// TIA Portal V16 program export: 6 tag tables, 0 data types, 9 data blocks, 25 code blocks (in call order from the OBs), 17 instance data blocks

VAR_GLOBAL   // PLC tag table "Analógicas"
   FQ301_MEDIDOR_CAUDAL AT %IW16 : Word;
   PC401_SENSOR_PRESSÃO AT %IW18 : Word;
END_VAR

VAR_GLOBAL   // PLC tag table "Default tag table"
   FirstScan AT %M1.0 : Bool;
   FALLING_EDGE_MAN_AUTO AT %M100.0 : Bool;
   RISING_EDGE_ETAPA_6 AT %M100.2 : Bool;
   FALLING_EDGE_BOT_EMERG AT %M100.5 : Bool;
   FALLIN_EDGE_BOT_EMERG_2 AT %M100.6 : Bool;
   FALLING_EDGE_ETAPA_6 AT %M100.7 : Bool;
   MBIT_DISP_1 AT %M101.0 : Bool;
   MBIT_DISP_2 AT %M101.1 : Bool;
   MBIT_DISP_3 AT %M101.2 : Bool;
   MBIT_DISP_4 AT %M101.3 : Bool;
   MBIT_DISP_5 AT %M101.4 : Bool;
   MBIT_DISP_6 AT %M101.5 : Bool;
   MBIT_DISP_7 AT %M101.6 : Bool;
   MBIT_DISP_8 AT %M101.7 : Bool;
   MBIT_DISP_9 AT %M102.0 : Bool;
   MBIT_DISP_10 AT %M102.1 : Bool;
   MBIT_DISP_11 AT %M102.2 : Bool;
   MBIT_DISP_12 AT %M102.3 : Bool;
   MBIT_DISP_13 AT %M102.4 : Bool;
   MBIT_DISP_14 AT %M102.5 : Bool;
   MBIT_DISP_15 AT %M102.6 : Bool;
   MBIT_DISP_16 AT %M102.7 : Bool;
   MBIT_DISP_DIF_3Q1_32 AT %M103.0 : Bool;
   MBIT_DISP_DIF_3Q3 AT %M103.1 : Bool;
   MBIT_DISP_DIF_4Q1_4Q2 AT %M103.2 : Bool;
   MBIT_FALHA_24VDC AT %M103.3 : Bool;
   MBIT_FALHA_220VAC AT %M103.4 : Bool;
   MBIT_FALHA_24VAC AT %M103.5 : Bool;
   RISING_EDGE_ETAPA_55 AT %M103.7 : Bool;
   RISING_EDGE_START_CICLO AT %M104.0 : Bool;
   Tag_1 AT %M200.0 : Bool;
END_VAR

VAR_GLOBAL   // PLC tag table "Estados_Componentes"
   BS001A_ON AT %I1.5 : Bool;
   BS001A_DISPARO AT %I2.0 : Bool;
   BS001B_ON AT %I2.1 : Bool;
   BS001B_DISPARO AT %I2.2 : Bool;
   XV102_ABERTA AT %I2.3 : Bool;
   XV102_FECHADA AT %I2.4 : Bool;
   XV101_ABERTA AT %I2.5 : Bool;
   MX201_ON AT %I2.6 : Bool;
   MX201_DISPARO AT %I2.7 : Bool;
   BH201_ON AT %I3.0 : Bool;
   BH201_DISPARO AT %I3.1 : Bool;
   MX301_ON AT %I3.2 : Bool;
   MX301_DISPARO AT %I3.3 : Bool;
   BM401_ON AT %I3.4 : Bool;
   BM401_DISPARO AT %I3.5 : Bool;
   BS501_ON AT %I3.6 : Bool;
   BS501_DISPARO AT %I3.7 : Bool;
   MX601_ON AT %I4.0 : Bool;
   MX601_DISPARO AT %I4.1 : Bool;
   BD601_ON AT %I4.2 : Bool;
   BD601_DISPARO AT %I4.3 : Bool;
   BD602_ON AT %I4.4 : Bool;
   BD602_DISPARO AT %I4.5 : Bool;
   MX603_ON AT %I4.6 : Bool;
   MX603_DISPARO AT %I4.7 : Bool;
   BD603_ON AT %I5.0 : Bool;
   BD603_DISPARO AT %I5.1 : Bool;
   MX604_ON AT %I5.2 : Bool;
   MX604_DISPARO AT %I5.3 : Bool;
   BD604_ON AT %I5.4 : Bool;
   BD604_DISPARO AT %I5.5 : Bool;
   MX605_ON AT %I5.6 : Bool;
   MX605_DISPARO AT %I5.7 : Bool;
   BD605_ON AT %I6.0 : Bool;
   BD605_DISPARO AT %I6.1 : Bool;
   BOT_EMERGÊNCIA AT %I6.2 : Bool;
   PH201_CONT_PH AT %I6.3 : Bool;
   PH301_CONT_PH AT %I6.4 : Bool;
   TEMPERATURA_ATINGIDA AT %I6.5 : Bool;
   RH201_CONT_REDOX AT %I6.6 : Bool;
END_VAR

VAR_GLOBAL   // PLC tag table "Falhas"
   DISPARO_DIF_3Q1_32 AT %I0.0 : Bool;
   DISPARO_DIFERENCIAL_3Q3 AT %I0.1 : Bool;
   DISPARO_DIFERENCIAL_4Q1_4Q2 AT %I0.2 : Bool;
   FALHA_24VDC AT %I0.3 : Bool;
   FALHA_220VAC AT %I0.4 : Bool;
   FALHA_24VAC AT %I0.5 : Bool;
END_VAR

VAR_GLOBAL   // PLC tag table "Níveis"
   LSH001_TK00 AT %I0.6 : Bool;
   LSL001_TK00 AT %I1.0 : Bool;
   LSH501_TK05 AT %I1.3 : Bool;
   LSL501_TK05 AT %I1.4 : Bool;
   LSH101_TK01 AT %I1.1 : Bool;
   LS201_TK02 AT %IW12 : Word;
   LS301_TK03 AT %IW14 : Word;
   LSL101_TK01 AT %I1.2 : Bool;
   LSM001_TK00 AT %I0.7 : Bool;
END_VAR

VAR_GLOBAL   // PLC tag table "Saídas"
   BS001A AT %Q0.0 : Bool;
   BS001B AT %Q0.1 : Bool;
   XV101 AT %Q3.3 : Bool;
   XV102 AT %Q3.4 : Bool;
   MX201 AT %Q0.4 : Bool;
   BH201 AT %Q0.5 : Bool;
   MX301 AT %Q0.6 : Bool;
   ALIM_BM401 AT %Q0.7 : Bool;
   LIGAR_BM401 AT %Q3.1 : Bool;
   BS501 AT %Q1.1 : Bool;
   MX601 AT %Q2.0 : Bool;
   BD601 AT %Q2.1 : Bool;
   BD602 AT %Q2.2 : Bool;
   MX603 AT %Q2.3 : Bool;
   BD603 AT %Q2.4 : Bool;
   MX604 AT %Q2.5 : Bool;
   BD604 AT %Q2.6 : Bool;
   MX605 AT %Q2.7 : Bool;
   BD605 AT %Q0.2 : Bool;
   ALARME AT %Q3.2 : Bool;
END_VAR

DATA_BLOCK "Alarmes"   // DB13
{ S7_Optimized_Access := 'TRUE' }
VERSION : 0.1
// stored: AutoNumber true, IsOnlyStoredInLoadMemory false, IsRetainMemResEnabled false, IsWriteProtectedInAS false, MemoryReserve 100
   VAR
      ALARMES_1 : Word;
      ALARMES_2 : Word;
      ALARME_DISPARO : Bool;
      PRESSÃO_MÁX : Bool;
      XV102_NÃO_ABRIU : Bool;
      XV102_NÃO_FECHOU : Bool;
   END_VAR
   VAR RETAIN
      TEMP_ABERT_XV102 : Time;
      TEMP_FECHO_XV102 : Time;
   END_VAR
BEGIN
END_DATA_BLOCK

DATA_BLOCK "Info_Ciclo"   // DB10
{ S7_Optimized_Access := 'TRUE' }
VERSION : 0.1
// stored: AutoNumber true, IsOnlyStoredInLoadMemory false, IsRetainMemResEnabled false, IsWriteProtectedInAS false, MemoryReserve 100
   VAR RETAIN
      LS101_SR : Bool;
   END_VAR
   VAR
      ESTADO_CICLO : Bool;
      CONTAGEM_CICLOS : Int;
      LIMITE_CONTAGEM : Bool;
   END_VAR
BEGIN
END_DATA_BLOCK

DATA_BLOCK "Analógicas"   // DB12
{ S7_Optimized_Access := 'TRUE' }
VERSION : 0.1
// stored: AutoNumber true, IsOnlyStoredInLoadMemory false, IsRetainMemResEnabled false, IsWriteProtectedInAS false, MemoryReserve 100
   VAR
      CAUDAL_FQ301 : Real;
      PRESSÃO_PC401 : Real;
   END_VAR
BEGIN
END_DATA_BLOCK

DATA_BLOCK "Estados_HMI_DB"   // DB15
{ S7_Optimized_Access := 'TRUE' }
VERSION : 0.1
// stored: AutoNumber true, IsOnlyStoredInLoadMemory false, IsRetainMemResEnabled false, IsWriteProtectedInAS false, MemoryReserve 100
   VAR
      MX201 : Bool;
      MX601 : Bool;
      XV101 : Bool;
      XV102 : Bool;
      BD601 : Bool;
      BD602 : Bool;
      BH201 : Bool;
      PH201 : Bool;
      RH201 : Bool;
      MX603 : Bool;
      BD603 : Bool;
      MX301 : Bool;
      PH301 : Bool;
      BM401 : Bool;
      MX604 : Bool;
      BD604 : Bool;
      MX605 : Bool;
      BD605 : Bool;
      BS001A : Bool;
      BS001B : Bool;
      BS501 : Bool;
      T_ATUAL_AREJAMENTO : Time;
      T_ATUAL_REDUÇÃO : Time;
      T_ATUAL_PRECIPITAÇÃO : Time;
      T_ATUAL_ALARME_PC401 : Time;
      T_ATUAL_COAG : Time;
      T_ATUAL_HISTERESE : Time;
   END_VAR
BEGIN
END_DATA_BLOCK

DATA_BLOCK "Inputs_HMI"   // DB14
{ S7_Optimized_Access := 'TRUE' }
VERSION : 0.1
// stored: AutoNumber true, IsOnlyStoredInLoadMemory false, IsRetainMemResEnabled false, IsWriteProtectedInAS false, MemoryReserve 100
   VAR RETAIN
      MODO_1 : Bool;
      MODO_2 : Bool;
   END_VAR
   VAR
      RESET_ALARME : Bool;
      START_CICLO : Bool;
   END_VAR
   VAR RETAIN
      MAN_AUTO : Bool;
   END_VAR
   VAR
      ON_OFF_MX201 : Bool;
      ON_OFF_MX301 : Bool;
      ON_OFF_MX601 : Bool;
      ON_OFF_MX603 : Bool;
      ON_OFF_MX604 : Bool;
      ON_OFF_MX605 : Bool;
      ON_OFF_BD601 : Bool;
      ON_OFF_BD602 : Bool;
      ON_OFF_BD603 : Bool;
      ON_OFF_BD604 : Bool;
      ON_OFF_BD605 : Bool;
      ON_OFF_BS001A : Bool;
      ON_OFF_BS001B : Bool;
      ON_OFF_BS501 : Bool;
      ON_OFF_BH201 : Bool;
      ON_OFF_BM401 : Bool;
      ON_OFF_XV101 : Bool;
      ON_OFF_XV102 : Bool;
   END_VAR
   VAR RETAIN
      TEMP_AREJAMENTO : Time := T#0m;
      TEMP_REDUÇÃO : Time := T#0m;
      TEMP_PRECIPITAÇÃO : Time := T#0m;
      TEMP_ALARME : Time := T#0m;
      TEMP_DOS_COAG : Time;
      HISTERESE : Time;
      SETPOINT_PC401 : Real;
      SP_LSH_TK02 : Real;
      SP_LSM_TK02 : Real;
      SP_LSL_TK02 : Real;
      SP_LSH_TK03 : Real;
      SP_LSM_TK03 : Real;
      SP_LSL_TK03 : Real;
   END_VAR
   VAR
      SALTAR_HISTERESE : Bool;
      RESET_CONT_CICLOS : Bool;
   END_VAR
   VAR RETAIN
      ENABLE_DISABLE_BD603 : Bool := true;
      SUSPENSÃO_CICLO_PRENSA : Bool;
      IGNORAR_LSH101_LSH501 : Bool;
   END_VAR
BEGIN
END_DATA_BLOCK

DATA_BLOCK "Níveis_TK02_TK03"   // DB11
{ S7_Optimized_Access := 'TRUE' }
VERSION : 0.1
// stored: AutoNumber true, IsOnlyStoredInLoadMemory false, IsRetainMemResEnabled false, IsWriteProtectedInAS false, MemoryReserve 100
   VAR
      LSH301 : Bool;
      LSM301 : Bool;
   END_VAR
   VAR RETAIN
      LSL301 : Bool;
   END_VAR
   VAR
      LSH201 : Bool;
      LSM201 : Bool;
      LSL201 : Bool;
      NÍVEL_EM_METROS_TK03 : Real;
      NÍVEL_EM_METROS_TK02 : Real;
   END_VAR
BEGIN
END_DATA_BLOCK

DATA_BLOCK "Etapas_Grafcet_1"   // DB4
{ S7_Optimized_Access := 'TRUE' }
VERSION : 0.1
// stored: AutoNumber true, IsOnlyStoredInLoadMemory false, IsRetainMemResEnabled false, IsWriteProtectedInAS false, MemoryReserve 100
   VAR RETAIN
      ETAPA_1 : Bool;
      ETAPA_2 : Bool;
      ETAPA_3 : Bool;
      ETAPA_4 : Bool;
      ETAPA_5 : Bool;
      ETAPA_6 : Bool;
      ETAPA_7 : Bool;
      ETAPA_8 : Bool;
      ETAPA_9 : Bool;
      ETAPA_33 : Bool;
      ETAPA_55 : Bool;
      RESET_ETAPA_1 : Bool;
      SUSPENSÃO_CICLO : Bool;
   END_VAR
BEGIN
END_DATA_BLOCK

DATA_BLOCK "Etapas_Grafcet_2"   // DB1
{ S7_Optimized_Access := 'TRUE' }
VERSION : 0.1
// stored: AutoNumber true, IsOnlyStoredInLoadMemory false, IsRetainMemResEnabled false, IsWriteProtectedInAS false, MemoryReserve 100
   VAR RETAIN
      ETAPA_10 : Bool;
      ETAPA_11 : Bool;
      ETAPA_12 : Bool;
      RESET_ETAPA_10 : Bool;
   END_VAR
BEGIN
END_DATA_BLOCK

DATA_BLOCK "Etapas_Grafcet_3"   // DB3
{ S7_Optimized_Access := 'TRUE' }
VERSION : 0.1
// stored: AutoNumber true, IsOnlyStoredInLoadMemory false, IsRetainMemResEnabled false, IsWriteProtectedInAS false, MemoryReserve 100
   VAR RETAIN
      ETAPA_13 : Bool;
      ETAPA_14 : Bool;
      ETAPA_15 : Bool;
      RESET_ETAPA_13 : Bool;
   END_VAR
BEGIN
END_DATA_BLOCK

ORGANIZATION_BLOCK "Main"   // OB1, LAD, ProgramCycle
TITLE = "Main Program Sweep (Cycle)"
{ S7_Optimized_Access := 'TRUE' }
VERSION : 0.1
// stored: AutoNumber true, IsIECCheckEnabled false, SetENOAutomatically false
BEGIN

REGION Network 1: Alimentação ao processo
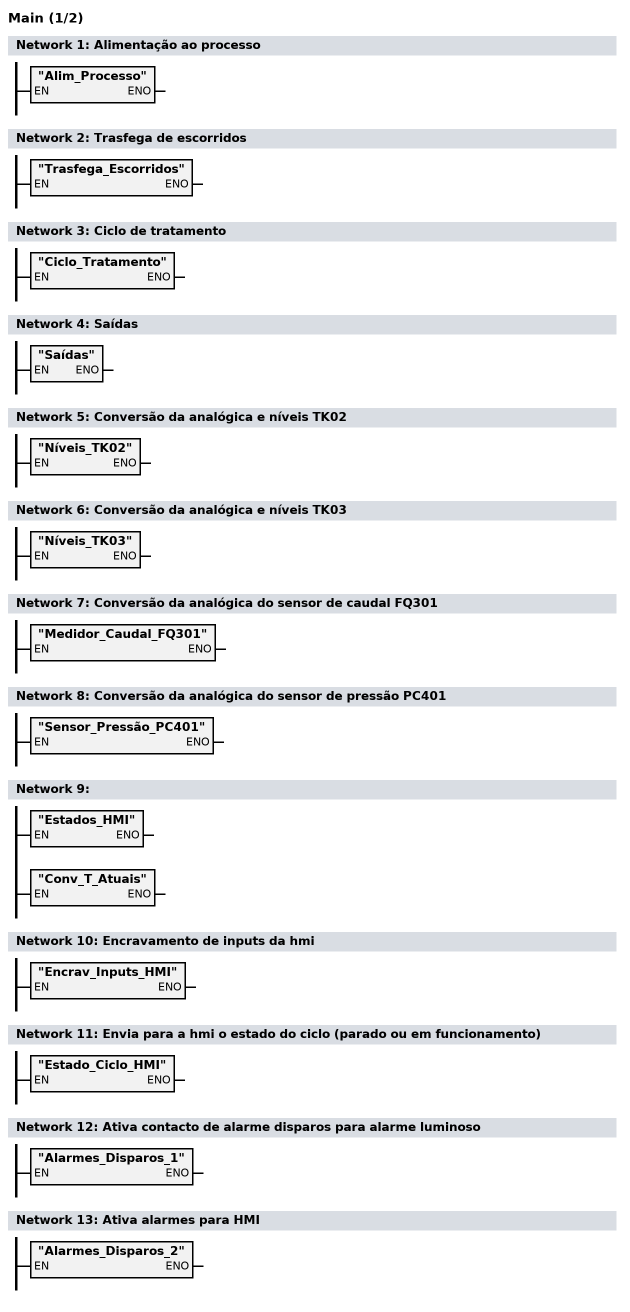
   RUNG wire#powerrail
      "Alim_Processo"()
   END_RUNG
   // the same network as SCL:
   "Alim_Processo"();
END_REGION

REGION Network 2: Trasfega de escorridos
   RUNG wire#powerrail
      "Trasfega_Escorridos"()
   END_RUNG
   // the same network as SCL:
   "Trasfega_Escorridos"();
END_REGION

REGION Network 3: Ciclo de tratamento
   RUNG wire#powerrail
      "Ciclo_Tratamento"()
   END_RUNG
   // the same network as SCL:
   "Ciclo_Tratamento"();
END_REGION

REGION Network 4: Saídas
   RUNG wire#powerrail
      "Saídas"()
   END_RUNG
   // the same network as SCL:
   "Saídas"();
END_REGION

REGION Network 5: Conversão da analógica e níveis TK02
   RUNG wire#powerrail
      "Níveis_TK02"()
   END_RUNG
   // the same network as SCL:
   "Níveis_TK02"();
END_REGION

REGION Network 6: Conversão da analógica e níveis TK03
   RUNG wire#powerrail
      "Níveis_TK03"()
   END_RUNG
   // the same network as SCL:
   "Níveis_TK03"();
END_REGION

REGION Network 7: Conversão da analógica do sensor de caudal FQ301
   RUNG wire#powerrail
      "Medidor_Caudal_FQ301"()
   END_RUNG
   // the same network as SCL:
   "Medidor_Caudal_FQ301"();
END_REGION

REGION Network 8: Conversão da analógica do sensor de pressão PC401
   RUNG wire#powerrail
      "Sensor_Pressão_PC401"()
   END_RUNG
   // the same network as SCL:
   "Sensor_Pressão_PC401"();
END_REGION

REGION Network 9
   RUNG wire#powerrail
      "Estados_HMI"()
   END_RUNG
   RUNG wire#powerrail
      "Conv_T_Atuais"()
   END_RUNG
   // the same network as SCL:
   "Estados_HMI"();
   "Conv_T_Atuais"();
END_REGION

REGION Network 10: Encravamento de inputs da hmi
   RUNG wire#powerrail
      "Encrav_Inputs_HMI"()
   END_RUNG
   // the same network as SCL:
   "Encrav_Inputs_HMI"();
END_REGION

REGION Network 11: Envia para a hmi o estado do ciclo (parado ou em funcionamento)
   RUNG wire#powerrail
      "Estado_Ciclo_HMI"()
   END_RUNG
   // the same network as SCL:
   "Estado_Ciclo_HMI"();
END_REGION

REGION Network 12: Ativa contacto de alarme disparos para alarme luminoso
   RUNG wire#powerrail
      "Alarmes_Disparos_1"()
   END_RUNG
   // the same network as SCL:
   "Alarmes_Disparos_1"();
END_REGION

REGION Network 13: Ativa alarmes para HMI
   RUNG wire#powerrail
      "Alarmes_Disparos_2"()
   END_RUNG
   // the same network as SCL:
   "Alarmes_Disparos_2"();
END_REGION

REGION Network 14: Alarme XV102 (não abriu/não fechou)
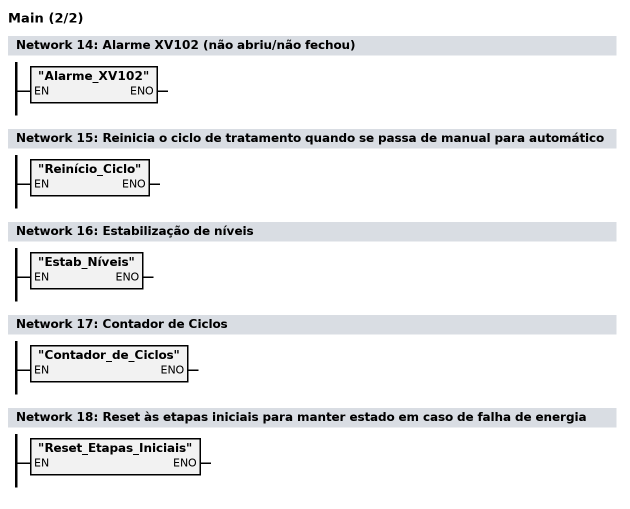
   RUNG wire#powerrail
      "Alarme_XV102"()
   END_RUNG
   // the same network as SCL:
   "Alarme_XV102"();
END_REGION

REGION Network 15: Reinicia o ciclo de tratamento quando se passa de manual para automático
   RUNG wire#powerrail
      "Reinício_Ciclo"()
   END_RUNG
   // the same network as SCL:
   "Reinício_Ciclo"();
END_REGION

REGION Network 16: Estabilização de níveis
   RUNG wire#powerrail
      "Estab_Níveis"()
   END_RUNG
   // the same network as SCL:
   "Estab_Níveis"();
END_REGION

REGION Network 17: Contador de Ciclos
   RUNG wire#powerrail
      "Contador_de_Ciclos"()
   END_RUNG
   // the same network as SCL:
   "Contador_de_Ciclos"();
END_REGION

REGION Network 18: Reset às etapas iniciais para manter estado em caso de falha de energia
   RUNG wire#powerrail
      "Reset_Etapas_Iniciais"()
   END_RUNG
   // the same network as SCL:
   "Reset_Etapas_Iniciais"();
END_REGION
END_ORGANIZATION_BLOCK

FUNCTION "Alim_Processo" : Void   // FC1, LAD
{ S7_Optimized_Access := 'TRUE' }
VERSION : 0.1
// stored: AutoNumber true, IsIECCheckEnabled false, SetENOAutomatically false, UDAEnableTagReadback false
BEGIN

REGION Network 1: Etapa 10 (INÍCIO)
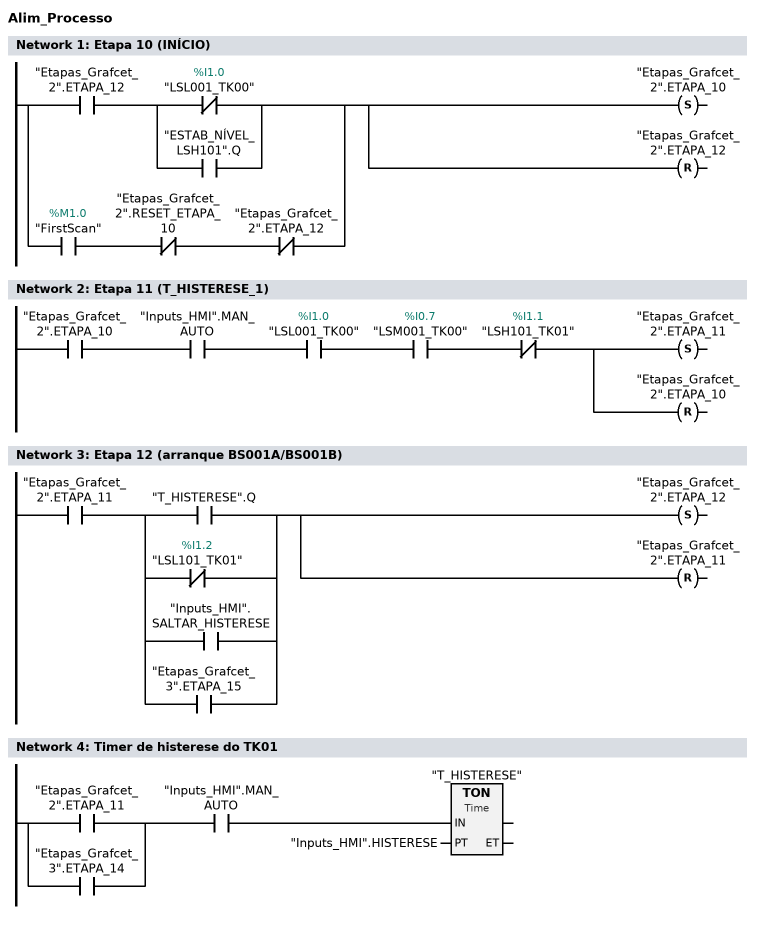
   RUNG wire#powerrail
      Contact( "Etapas_Grafcet_2".ETAPA_12 )
      wire#w1
      I_Contact( "LSL001_TK00" )
      wire#w2
      S_Coil( "Etapas_Grafcet_2".ETAPA_10 )
   END_RUNG
   RUNG wire#w1
      Contact( "ESTAB_NÍVEL_LSH101".Q )
   END_RUNG wire#w2
   RUNG wire#powerrail
      Contact( "FirstScan" )
      I_Contact( "Etapas_Grafcet_2".RESET_ETAPA_10 )
      I_Contact( "Etapas_Grafcet_2".ETAPA_12 )
   END_RUNG wire#w2
   RUNG wire#w2
      R_Coil( "Etapas_Grafcet_2".ETAPA_12 )
   END_RUNG
   // the same network as SCL:
   IF ("Etapas_Grafcet_2".ETAPA_12 AND (NOT "LSL001_TK00" OR "ESTAB_NÍVEL_LSH101".Q)) OR ("FirstScan" AND NOT "Etapas_Grafcet_2".RESET_ETAPA_10 AND NOT "Etapas_Grafcet_2".ETAPA_12) THEN
       "Etapas_Grafcet_2".ETAPA_10 := TRUE;
       "Etapas_Grafcet_2".ETAPA_12 := FALSE;
   END_IF;
END_REGION

REGION Network 2: Etapa 11 (T_HISTERESE_1)
   RUNG wire#powerrail
      Contact( "Etapas_Grafcet_2".ETAPA_10 )
      Contact( "Inputs_HMI".MAN_AUTO )
      Contact( "LSL001_TK00" )
      Contact( "LSM001_TK00" )
      I_Contact( "LSH101_TK01" )
      wire#w1
      S_Coil( "Etapas_Grafcet_2".ETAPA_11 )
   END_RUNG
   RUNG wire#w1
      R_Coil( "Etapas_Grafcet_2".ETAPA_10 )
   END_RUNG
   // the same network as SCL:
   IF "Etapas_Grafcet_2".ETAPA_10 AND "Inputs_HMI".MAN_AUTO AND "LSL001_TK00" AND "LSM001_TK00" AND NOT "LSH101_TK01" THEN
       "Etapas_Grafcet_2".ETAPA_11 := TRUE;
       "Etapas_Grafcet_2".ETAPA_10 := FALSE;
   END_IF;
END_REGION

REGION Network 3: Etapa 12 (arranque BS001A/BS001B)
   RUNG wire#powerrail
      Contact( "Etapas_Grafcet_2".ETAPA_11 )
      wire#w1
      Contact( "T_HISTERESE".Q )
      wire#w2
      S_Coil( "Etapas_Grafcet_2".ETAPA_12 )
   END_RUNG
   RUNG wire#w1
      I_Contact( "LSL101_TK01" )
   END_RUNG wire#w2
   RUNG wire#w1
      Contact( "Inputs_HMI".SALTAR_HISTERESE )
   END_RUNG wire#w2
   RUNG wire#w1
      Contact( "Etapas_Grafcet_3".ETAPA_15 )
   END_RUNG wire#w2
   RUNG wire#w2
      R_Coil( "Etapas_Grafcet_2".ETAPA_11 )
   END_RUNG
   // the same network as SCL:
   IF "Etapas_Grafcet_2".ETAPA_11 AND ("T_HISTERESE".Q OR NOT "LSL101_TK01" OR "Inputs_HMI".SALTAR_HISTERESE OR "Etapas_Grafcet_3".ETAPA_15) THEN
       "Etapas_Grafcet_2".ETAPA_12 := TRUE;
       "Etapas_Grafcet_2".ETAPA_11 := FALSE;
   END_IF;
END_REGION

REGION Network 4: Timer de histerese do TK01
   RUNG wire#powerrail
      Contact( "Etapas_Grafcet_2".ETAPA_11 )
      wire#w1
      Contact( "Inputs_HMI".MAN_AUTO )
      { S7_Templates := "time_type := Time" } "T_HISTERESE".TON(pt := "Inputs_HMI".HISTERESE, et =>)
   END_RUNG
   RUNG wire#powerrail
      Contact( "Etapas_Grafcet_3".ETAPA_14 )
   END_RUNG wire#w1
   // the same network as SCL:
   "T_HISTERESE".TON(IN := ("Etapas_Grafcet_2".ETAPA_11 OR "Etapas_Grafcet_3".ETAPA_14) AND "Inputs_HMI".MAN_AUTO,
                     PT := "Inputs_HMI".HISTERESE);
END_REGION
END_FUNCTION

FUNCTION "Trasfega_Escorridos" : Void   // FC3, LAD
{ S7_Optimized_Access := 'TRUE' }
VERSION : 0.1
// stored: AutoNumber true, IsIECCheckEnabled false, SetENOAutomatically false, UDAEnableTagReadback false
BEGIN

REGION Network 1: Etapa 13 (INÍCIO)
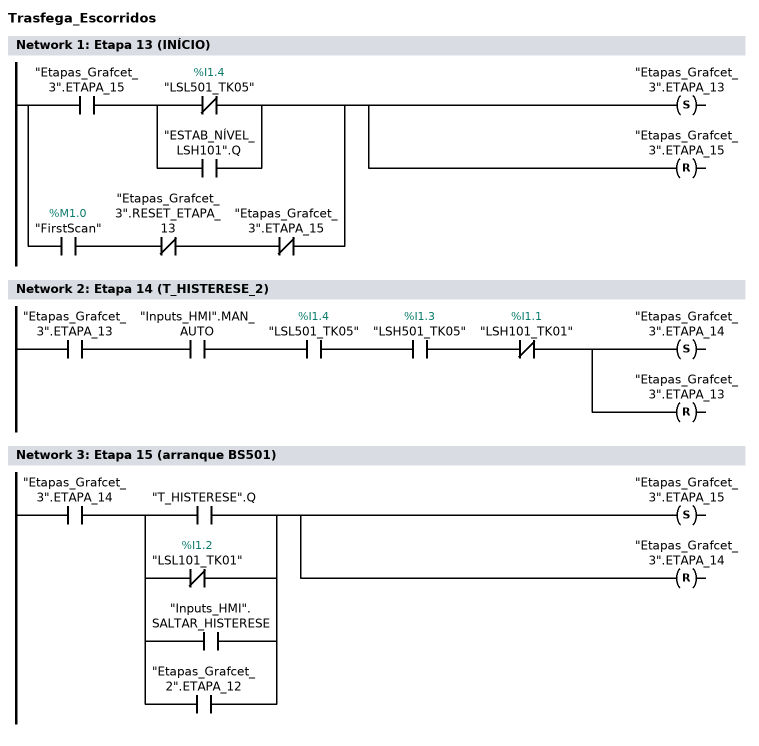
   RUNG wire#powerrail
      Contact( "Etapas_Grafcet_3".ETAPA_15 )
      wire#w1
      I_Contact( "LSL501_TK05" )
      wire#w2
      S_Coil( "Etapas_Grafcet_3".ETAPA_13 )
   END_RUNG
   RUNG wire#w1
      Contact( "ESTAB_NÍVEL_LSH101".Q )
   END_RUNG wire#w2
   RUNG wire#powerrail
      Contact( "FirstScan" )
      I_Contact( "Etapas_Grafcet_3".RESET_ETAPA_13 )
      I_Contact( "Etapas_Grafcet_3".ETAPA_15 )
   END_RUNG wire#w2
   RUNG wire#w2
      R_Coil( "Etapas_Grafcet_3".ETAPA_15 )
   END_RUNG
   // the same network as SCL:
   IF ("Etapas_Grafcet_3".ETAPA_15 AND (NOT "LSL501_TK05" OR "ESTAB_NÍVEL_LSH101".Q)) OR ("FirstScan" AND NOT "Etapas_Grafcet_3".RESET_ETAPA_13 AND NOT "Etapas_Grafcet_3".ETAPA_15) THEN
       "Etapas_Grafcet_3".ETAPA_13 := TRUE;
       "Etapas_Grafcet_3".ETAPA_15 := FALSE;
   END_IF;
END_REGION

REGION Network 2: Etapa 14 (T_HISTERESE_2)
   RUNG wire#powerrail
      Contact( "Etapas_Grafcet_3".ETAPA_13 )
      Contact( "Inputs_HMI".MAN_AUTO )
      Contact( "LSL501_TK05" )
      Contact( "LSH501_TK05" )
      I_Contact( "LSH101_TK01" )
      wire#w1
      S_Coil( "Etapas_Grafcet_3".ETAPA_14 )
   END_RUNG
   RUNG wire#w1
      R_Coil( "Etapas_Grafcet_3".ETAPA_13 )
   END_RUNG
   // the same network as SCL:
   IF "Etapas_Grafcet_3".ETAPA_13 AND "Inputs_HMI".MAN_AUTO AND "LSL501_TK05" AND "LSH501_TK05" AND NOT "LSH101_TK01" THEN
       "Etapas_Grafcet_3".ETAPA_14 := TRUE;
       "Etapas_Grafcet_3".ETAPA_13 := FALSE;
   END_IF;
END_REGION

REGION Network 3: Etapa 15 (arranque BS501)
   RUNG wire#powerrail
      Contact( "Etapas_Grafcet_3".ETAPA_14 )
      wire#w1
      Contact( "T_HISTERESE".Q )
      wire#w2
      S_Coil( "Etapas_Grafcet_3".ETAPA_15 )
   END_RUNG
   RUNG wire#w1
      I_Contact( "LSL101_TK01" )
   END_RUNG wire#w2
   RUNG wire#w1
      Contact( "Inputs_HMI".SALTAR_HISTERESE )
   END_RUNG wire#w2
   RUNG wire#w1
      Contact( "Etapas_Grafcet_2".ETAPA_12 )
   END_RUNG wire#w2
   RUNG wire#w2
      R_Coil( "Etapas_Grafcet_3".ETAPA_14 )
   END_RUNG
   // the same network as SCL:
   IF "Etapas_Grafcet_3".ETAPA_14 AND ("T_HISTERESE".Q OR NOT "LSL101_TK01" OR "Inputs_HMI".SALTAR_HISTERESE OR "Etapas_Grafcet_2".ETAPA_12) THEN
       "Etapas_Grafcet_3".ETAPA_15 := TRUE;
       "Etapas_Grafcet_3".ETAPA_14 := FALSE;
   END_IF;
END_REGION
END_FUNCTION

FUNCTION "Ciclo_Tratamento" : Void   // FC4, LAD
{ S7_Optimized_Access := 'TRUE' }
VERSION : 0.1
// stored: AutoNumber true, IsIECCheckEnabled false, SetENOAutomatically false, UDAEnableTagReadback false
   VAR_TEMP   // added for the SCL form of the ladder/FBD networks
      _w1 : Bool;
      _w2 : Bool;
   END_VAR
BEGIN

REGION Network 1: Etapa 1 (INÍCIO)
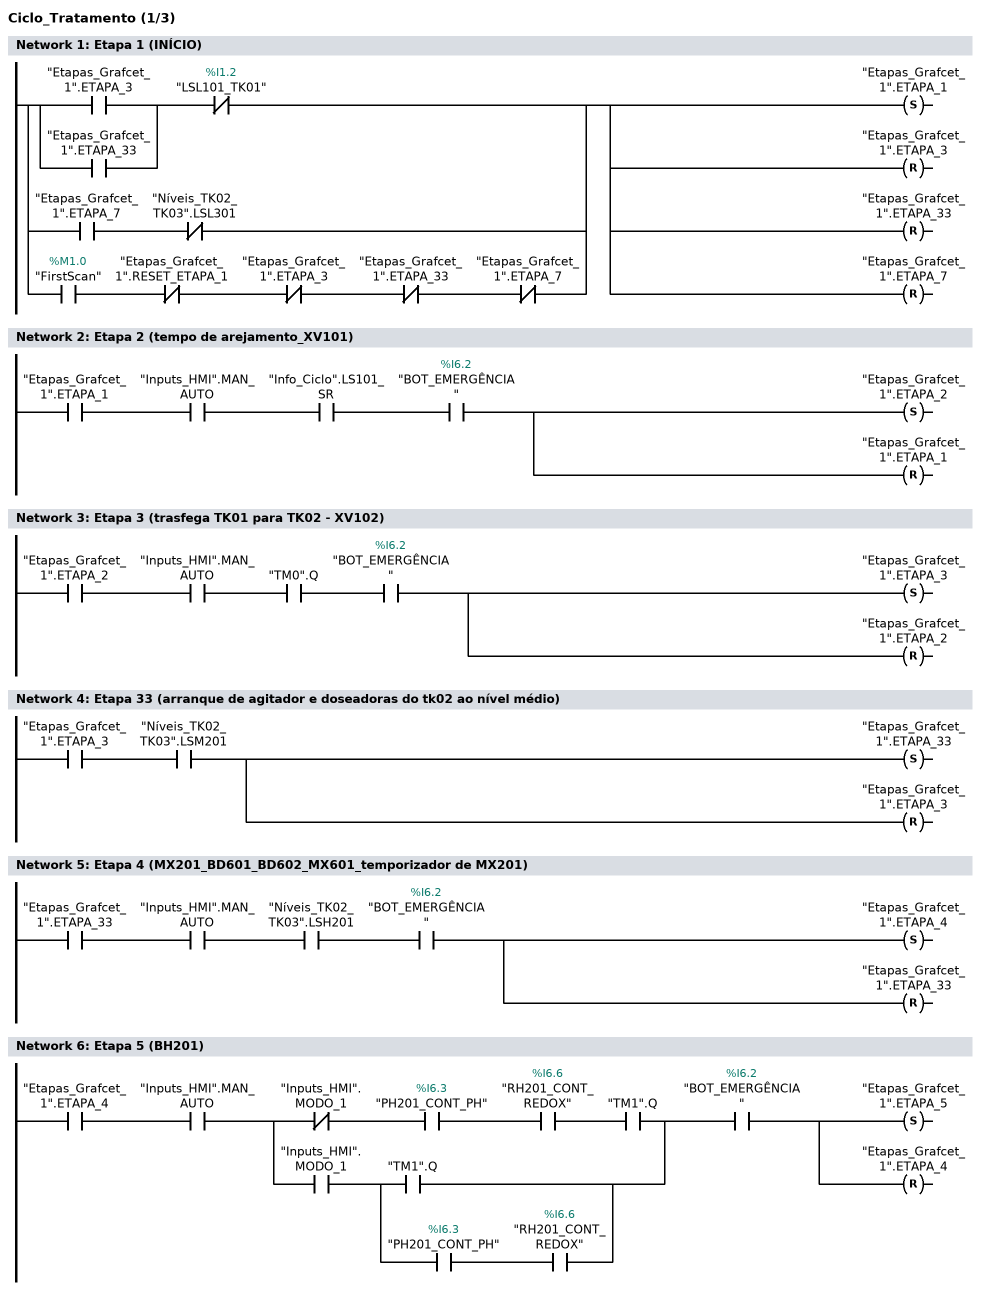
   RUNG wire#powerrail
      Contact( "Etapas_Grafcet_1".ETAPA_3 )
      wire#w1
      I_Contact( "LSL101_TK01" )
      wire#w2
      S_Coil( "Etapas_Grafcet_1".ETAPA_1 )
   END_RUNG
   RUNG wire#powerrail
      Contact( "Etapas_Grafcet_1".ETAPA_33 )
   END_RUNG wire#w1
   RUNG wire#powerrail
      Contact( "Etapas_Grafcet_1".ETAPA_7 )
      I_Contact( "Níveis_TK02_TK03".LSL301 )
   END_RUNG wire#w2
   RUNG wire#powerrail
      Contact( "FirstScan" )
      I_Contact( "Etapas_Grafcet_1".RESET_ETAPA_1 )
      I_Contact( "Etapas_Grafcet_1".ETAPA_3 )
      I_Contact( "Etapas_Grafcet_1".ETAPA_33 )
      I_Contact( "Etapas_Grafcet_1".ETAPA_7 )
   END_RUNG wire#w2
   RUNG wire#w2
      R_Coil( "Etapas_Grafcet_1".ETAPA_3 )
   END_RUNG
   RUNG wire#w2
      R_Coil( "Etapas_Grafcet_1".ETAPA_33 )
   END_RUNG
   RUNG wire#w2
      R_Coil( "Etapas_Grafcet_1".ETAPA_7 )
   END_RUNG
   // the same network as SCL:
   IF (("Etapas_Grafcet_1".ETAPA_3 OR "Etapas_Grafcet_1".ETAPA_33) AND NOT "LSL101_TK01") OR ("Etapas_Grafcet_1".ETAPA_7 AND NOT "Níveis_TK02_TK03".LSL301) OR ("FirstScan" AND NOT "Etapas_Grafcet_1".RESET_ETAPA_1 AND NOT "Etapas_Grafcet_1".ETAPA_3 AND NOT "Etapas_Grafcet_1".ETAPA_33 AND NOT "Etapas_Grafcet_1".ETAPA_7) THEN
       "Etapas_Grafcet_1".ETAPA_1 := TRUE;
   END_IF;
   #_w1 := (("Etapas_Grafcet_1".ETAPA_3 OR "Etapas_Grafcet_1".ETAPA_33) AND NOT "LSL101_TK01") OR ("Etapas_Grafcet_1".ETAPA_7 AND NOT "Níveis_TK02_TK03".LSL301) OR ("FirstScan" AND NOT "Etapas_Grafcet_1".RESET_ETAPA_1 AND NOT "Etapas_Grafcet_1".ETAPA_3 AND NOT "Etapas_Grafcet_1".ETAPA_33 AND NOT "Etapas_Grafcet_1".ETAPA_7);
   IF #_w1 THEN
       "Etapas_Grafcet_1".ETAPA_3 := FALSE;
       "Etapas_Grafcet_1".ETAPA_33 := FALSE;
       "Etapas_Grafcet_1".ETAPA_7 := FALSE;
   END_IF;
END_REGION

REGION Network 2: Etapa 2 (tempo de arejamento_XV101)
   RUNG wire#powerrail
      Contact( "Etapas_Grafcet_1".ETAPA_1 )
      Contact( "Inputs_HMI".MAN_AUTO )
      Contact( "Info_Ciclo".LS101_SR )
      Contact( "BOT_EMERGÊNCIA" )
      wire#w1
      S_Coil( "Etapas_Grafcet_1".ETAPA_2 )
   END_RUNG
   RUNG wire#w1
      R_Coil( "Etapas_Grafcet_1".ETAPA_1 )
   END_RUNG
   // the same network as SCL:
   IF "Etapas_Grafcet_1".ETAPA_1 AND "Inputs_HMI".MAN_AUTO AND "Info_Ciclo".LS101_SR AND "BOT_EMERGÊNCIA" THEN
       "Etapas_Grafcet_1".ETAPA_2 := TRUE;
       "Etapas_Grafcet_1".ETAPA_1 := FALSE;
   END_IF;
END_REGION

REGION Network 3: Etapa 3 (trasfega TK01 para TK02 - XV102)
   RUNG wire#powerrail
      Contact( "Etapas_Grafcet_1".ETAPA_2 )
      Contact( "Inputs_HMI".MAN_AUTO )
      Contact( "TM0".Q )
      Contact( "BOT_EMERGÊNCIA" )
      wire#w1
      S_Coil( "Etapas_Grafcet_1".ETAPA_3 )
   END_RUNG
   RUNG wire#w1
      R_Coil( "Etapas_Grafcet_1".ETAPA_2 )
   END_RUNG
   // the same network as SCL:
   IF "Etapas_Grafcet_1".ETAPA_2 AND "Inputs_HMI".MAN_AUTO AND "TM0".Q AND "BOT_EMERGÊNCIA" THEN
       "Etapas_Grafcet_1".ETAPA_3 := TRUE;
       "Etapas_Grafcet_1".ETAPA_2 := FALSE;
   END_IF;
END_REGION

REGION Network 4: Etapa 33 (arranque de agitador e doseadoras do tk02 ao nível médio)
   RUNG wire#powerrail
      Contact( "Etapas_Grafcet_1".ETAPA_3 )
      Contact( "Níveis_TK02_TK03".LSM201 )
      wire#w1
      S_Coil( "Etapas_Grafcet_1".ETAPA_33 )
   END_RUNG
   RUNG wire#w1
      R_Coil( "Etapas_Grafcet_1".ETAPA_3 )
   END_RUNG
   // the same network as SCL:
   IF "Etapas_Grafcet_1".ETAPA_3 AND "Níveis_TK02_TK03".LSM201 THEN
       "Etapas_Grafcet_1".ETAPA_33 := TRUE;
       "Etapas_Grafcet_1".ETAPA_3 := FALSE;
   END_IF;
END_REGION

REGION Network 5: Etapa 4 (MX201_BD601_BD602_MX601_temporizador de MX201)
   RUNG wire#powerrail
      Contact( "Etapas_Grafcet_1".ETAPA_33 )
      Contact( "Inputs_HMI".MAN_AUTO )
      Contact( "Níveis_TK02_TK03".LSH201 )
      Contact( "BOT_EMERGÊNCIA" )
      wire#w1
      S_Coil( "Etapas_Grafcet_1".ETAPA_4 )
   END_RUNG
   RUNG wire#w1
      R_Coil( "Etapas_Grafcet_1".ETAPA_33 )
   END_RUNG
   // the same network as SCL:
   IF "Etapas_Grafcet_1".ETAPA_33 AND "Inputs_HMI".MAN_AUTO AND "Níveis_TK02_TK03".LSH201 AND "BOT_EMERGÊNCIA" THEN
       "Etapas_Grafcet_1".ETAPA_4 := TRUE;
       "Etapas_Grafcet_1".ETAPA_33 := FALSE;
   END_IF;
END_REGION

REGION Network 6: Etapa 5 (BH201)
   RUNG wire#powerrail
      Contact( "Etapas_Grafcet_1".ETAPA_4 )
      Contact( "Inputs_HMI".MAN_AUTO )
      wire#w1
      I_Contact( "Inputs_HMI".MODO_1 )
      Contact( "PH201_CONT_PH" )
      Contact( "RH201_CONT_REDOX" )
      Contact( "TM1".Q )
      wire#w2
      Contact( "BOT_EMERGÊNCIA" )
      wire#w4
      S_Coil( "Etapas_Grafcet_1".ETAPA_5 )
   END_RUNG
   RUNG wire#w1
      Contact( "Inputs_HMI".MODO_1 )
      wire#w3
      Contact( "TM1".Q )
   END_RUNG wire#w2
   RUNG wire#w3
      Contact( "PH201_CONT_PH" )
      Contact( "RH201_CONT_REDOX" )
   END_RUNG wire#w2
   RUNG wire#w4
      R_Coil( "Etapas_Grafcet_1".ETAPA_4 )
   END_RUNG
   // the same network as SCL:
   IF "Etapas_Grafcet_1".ETAPA_4 AND "Inputs_HMI".MAN_AUTO AND ((NOT "Inputs_HMI".MODO_1 AND "PH201_CONT_PH" AND "RH201_CONT_REDOX" AND "TM1".Q) OR ("Inputs_HMI".MODO_1 AND ("TM1".Q OR ("PH201_CONT_PH" AND "RH201_CONT_REDOX")))) AND "BOT_EMERGÊNCIA" THEN
       "Etapas_Grafcet_1".ETAPA_5 := TRUE;
       "Etapas_Grafcet_1".ETAPA_4 := FALSE;
   END_IF;
END_REGION

REGION Network 7: Etapa 55 (arranque de agitador e doseadoras do tk03 ao nível médio)
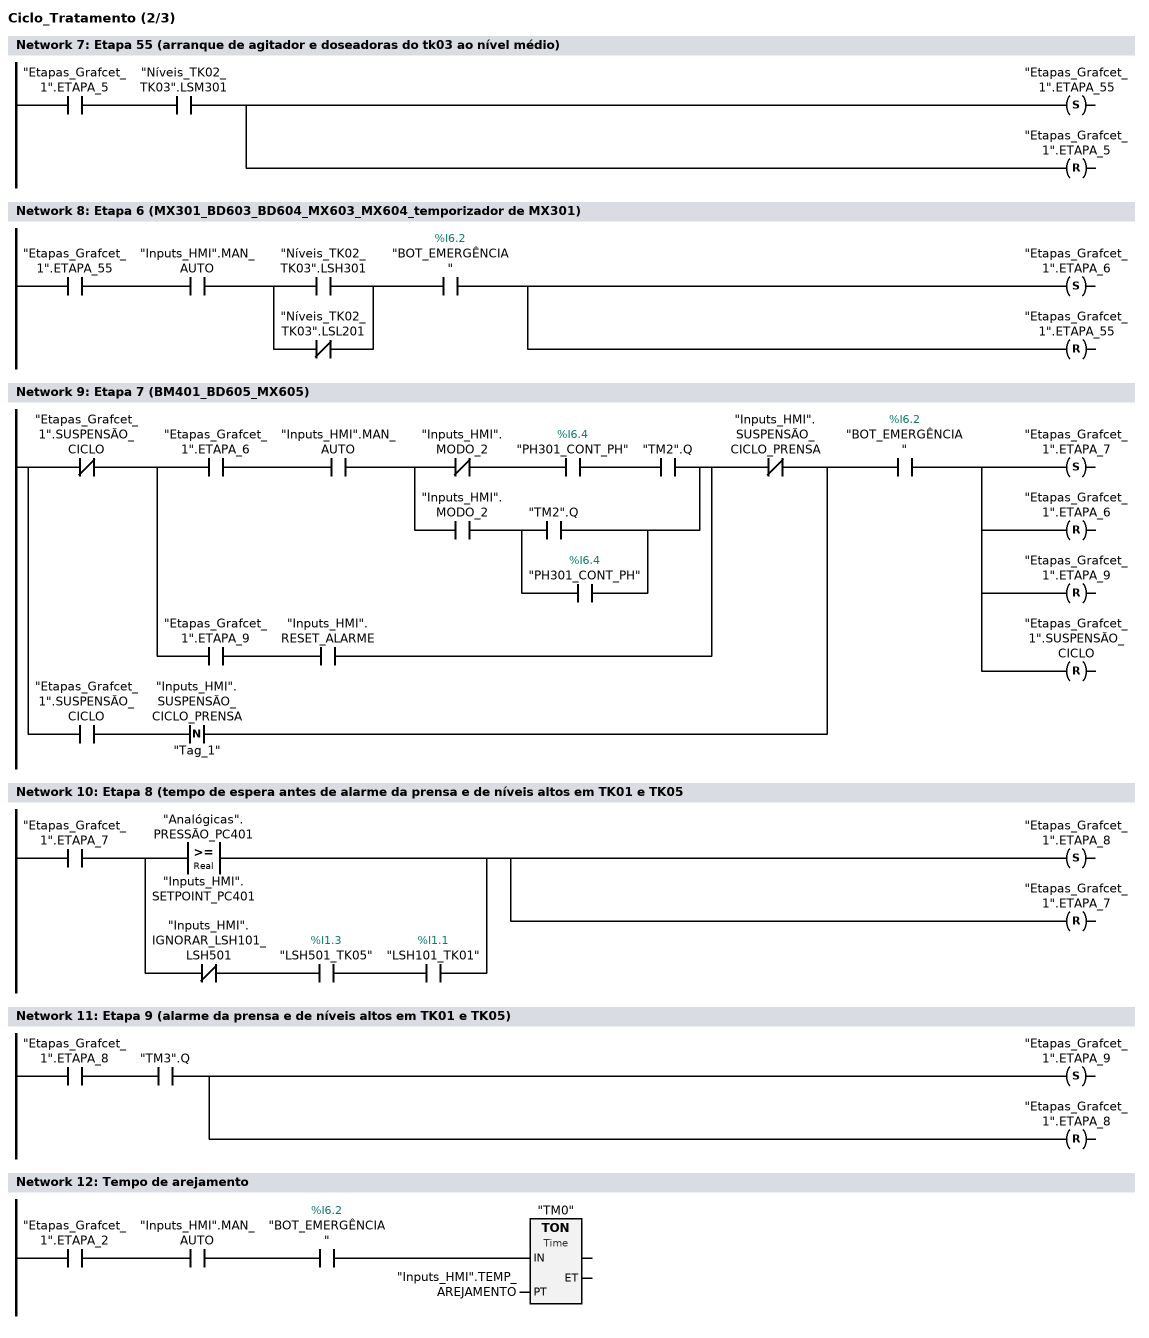
   RUNG wire#powerrail
      Contact( "Etapas_Grafcet_1".ETAPA_5 )
      Contact( "Níveis_TK02_TK03".LSM301 )
      wire#w1
      S_Coil( "Etapas_Grafcet_1".ETAPA_55 )
   END_RUNG
   RUNG wire#w1
      R_Coil( "Etapas_Grafcet_1".ETAPA_5 )
   END_RUNG
   // the same network as SCL:
   IF "Etapas_Grafcet_1".ETAPA_5 AND "Níveis_TK02_TK03".LSM301 THEN
       "Etapas_Grafcet_1".ETAPA_55 := TRUE;
       "Etapas_Grafcet_1".ETAPA_5 := FALSE;
   END_IF;
END_REGION

REGION Network 8: Etapa 6 (MX301_BD603_BD604_MX603_MX604_temporizador de MX301)
   RUNG wire#powerrail
      Contact( "Etapas_Grafcet_1".ETAPA_55 )
      Contact( "Inputs_HMI".MAN_AUTO )
      wire#w1
      Contact( "Níveis_TK02_TK03".LSH301 )
      wire#w2
      Contact( "BOT_EMERGÊNCIA" )
      wire#w3
      S_Coil( "Etapas_Grafcet_1".ETAPA_6 )
   END_RUNG
   RUNG wire#w1
      I_Contact( "Níveis_TK02_TK03".LSL201 )
   END_RUNG wire#w2
   RUNG wire#w3
      R_Coil( "Etapas_Grafcet_1".ETAPA_55 )
   END_RUNG
   // the same network as SCL:
   IF "Etapas_Grafcet_1".ETAPA_55 AND "Inputs_HMI".MAN_AUTO AND ("Níveis_TK02_TK03".LSH301 OR NOT "Níveis_TK02_TK03".LSL201) AND "BOT_EMERGÊNCIA" THEN
       "Etapas_Grafcet_1".ETAPA_6 := TRUE;
       "Etapas_Grafcet_1".ETAPA_55 := FALSE;
   END_IF;
END_REGION

REGION Network 9: Etapa 7 (BM401_BD605_MX605)
   RUNG wire#powerrail
      I_Contact( "Etapas_Grafcet_1".SUSPENSÃO_CICLO )
      wire#w1
      Contact( "Etapas_Grafcet_1".ETAPA_6 )
      Contact( "Inputs_HMI".MAN_AUTO )
      wire#w2
      I_Contact( "Inputs_HMI".MODO_2 )
      Contact( "PH301_CONT_PH" )
      Contact( "TM2".Q )
      wire#w3
      I_Contact( "Inputs_HMI".SUSPENSÃO_CICLO_PRENSA )
      wire#w5
      Contact( "BOT_EMERGÊNCIA" )
      wire#w6
      S_Coil( "Etapas_Grafcet_1".ETAPA_7 )
   END_RUNG
   RUNG wire#w2
      Contact( "Inputs_HMI".MODO_2 )
      wire#w4
      Contact( "TM2".Q )
   END_RUNG wire#w3
   RUNG wire#w4
      Contact( "PH301_CONT_PH" )
   END_RUNG wire#w3
   RUNG wire#w1
      Contact( "Etapas_Grafcet_1".ETAPA_9 )
      Contact( "Inputs_HMI".RESET_ALARME )
   END_RUNG wire#w3
   RUNG wire#powerrail
      Contact( "Etapas_Grafcet_1".SUSPENSÃO_CICLO )
      N_Contact(operand := "Inputs_HMI".SUSPENSÃO_CICLO_PRENSA, bit := "Tag_1")
   END_RUNG wire#w5
   RUNG wire#w6
      R_Coil( "Etapas_Grafcet_1".ETAPA_6 )
   END_RUNG
   RUNG wire#w6
      R_Coil( "Etapas_Grafcet_1".ETAPA_9 )
   END_RUNG
   RUNG wire#w6
      R_Coil( "Etapas_Grafcet_1".SUSPENSÃO_CICLO )
   END_RUNG
   // the same network as SCL:
   #_w1 := "Etapas_Grafcet_1".SUSPENSÃO_CICLO AND NOT "Inputs_HMI".SUSPENSÃO_CICLO_PRENSA AND "Tag_1";   // falling edge of "Inputs_HMI".SUSPENSÃO_CICLO_PRENSA
   "Tag_1" := "Inputs_HMI".SUSPENSÃO_CICLO_PRENSA;
   IF ((NOT "Etapas_Grafcet_1".SUSPENSÃO_CICLO AND (("Etapas_Grafcet_1".ETAPA_6 AND "Inputs_HMI".MAN_AUTO AND ((NOT "Inputs_HMI".MODO_2 AND "PH301_CONT_PH" AND "TM2".Q) OR ("Inputs_HMI".MODO_2 AND ("TM2".Q OR "PH301_CONT_PH")))) OR ("Etapas_Grafcet_1".ETAPA_9 AND "Inputs_HMI".RESET_ALARME)) AND NOT "Inputs_HMI".SUSPENSÃO_CICLO_PRENSA) OR #_w1) AND "BOT_EMERGÊNCIA" THEN
       "Etapas_Grafcet_1".ETAPA_7 := TRUE;
   END_IF;
   #_w2 := ((NOT "Etapas_Grafcet_1".SUSPENSÃO_CICLO AND (("Etapas_Grafcet_1".ETAPA_6 AND "Inputs_HMI".MAN_AUTO AND ((NOT "Inputs_HMI".MODO_2 AND "PH301_CONT_PH" AND "TM2".Q) OR ("Inputs_HMI".MODO_2 AND ("TM2".Q OR "PH301_CONT_PH")))) OR ("Etapas_Grafcet_1".ETAPA_9 AND "Inputs_HMI".RESET_ALARME)) AND NOT "Inputs_HMI".SUSPENSÃO_CICLO_PRENSA) OR #_w1) AND "BOT_EMERGÊNCIA";
   IF #_w2 THEN
       "Etapas_Grafcet_1".ETAPA_6 := FALSE;
       "Etapas_Grafcet_1".ETAPA_9 := FALSE;
       "Etapas_Grafcet_1".SUSPENSÃO_CICLO := FALSE;
   END_IF;
END_REGION

REGION Network 10: Etapa 8 (tempo de espera antes de alarme da prensa e de níveis altos em TK01 e TK05
   RUNG wire#powerrail
      Contact( "Etapas_Grafcet_1".ETAPA_7 )
      wire#w1
      { S7_Templates := "SrcType := Real" } GE_Contact(in1 := "Analógicas".PRESSÃO_PC401, in2 := "Inputs_HMI".SETPOINT_PC401)
      wire#w2
      S_Coil( "Etapas_Grafcet_1".ETAPA_8 )
   END_RUNG
   RUNG wire#w1
      I_Contact( "Inputs_HMI".IGNORAR_LSH101_LSH501 )
      Contact( "LSH501_TK05" )
      Contact( "LSH101_TK01" )
   END_RUNG wire#w2
   RUNG wire#w2
      R_Coil( "Etapas_Grafcet_1".ETAPA_7 )
   END_RUNG
   // the same network as SCL:
   IF "Etapas_Grafcet_1".ETAPA_7 AND (("Analógicas".PRESSÃO_PC401 >= "Inputs_HMI".SETPOINT_PC401) OR (NOT "Inputs_HMI".IGNORAR_LSH101_LSH501 AND "LSH501_TK05" AND "LSH101_TK01")) THEN
       "Etapas_Grafcet_1".ETAPA_8 := TRUE;
       "Etapas_Grafcet_1".ETAPA_7 := FALSE;
   END_IF;
END_REGION

REGION Network 11: Etapa 9 (alarme da prensa e de níveis altos em TK01 e TK05)
   RUNG wire#powerrail
      Contact( "Etapas_Grafcet_1".ETAPA_8 )
      Contact( "TM3".Q )
      wire#w1
      S_Coil( "Etapas_Grafcet_1".ETAPA_9 )
   END_RUNG
   RUNG wire#w1
      R_Coil( "Etapas_Grafcet_1".ETAPA_8 )
   END_RUNG
   // the same network as SCL:
   IF "Etapas_Grafcet_1".ETAPA_8 AND "TM3".Q THEN
       "Etapas_Grafcet_1".ETAPA_9 := TRUE;
       "Etapas_Grafcet_1".ETAPA_8 := FALSE;
   END_IF;
END_REGION

REGION Network 12: Tempo de arejamento
   RUNG wire#powerrail
      Contact( "Etapas_Grafcet_1".ETAPA_2 )
      Contact( "Inputs_HMI".MAN_AUTO )
      Contact( "BOT_EMERGÊNCIA" )
      { S7_Templates := "time_type := Time" } "TM0".TON(pt := "Inputs_HMI".TEMP_AREJAMENTO, et =>)
   END_RUNG
   // the same network as SCL:
   "TM0".TON(IN := "Etapas_Grafcet_1".ETAPA_2 AND "Inputs_HMI".MAN_AUTO AND "BOT_EMERGÊNCIA",
             PT := "Inputs_HMI".TEMP_AREJAMENTO);
END_REGION

REGION Network 13: Etapa Suspensão Ciclo
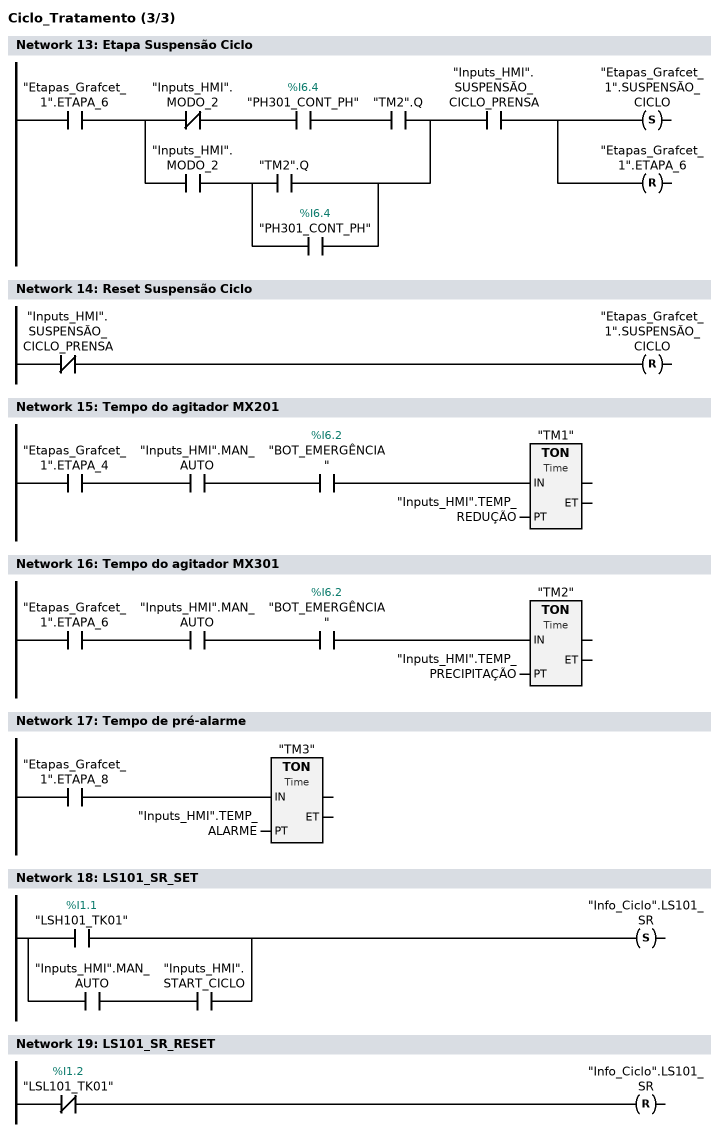
   RUNG wire#powerrail
      Contact( "Etapas_Grafcet_1".ETAPA_6 )
      wire#w1
      I_Contact( "Inputs_HMI".MODO_2 )
      Contact( "PH301_CONT_PH" )
      Contact( "TM2".Q )
      wire#w2
      Contact( "Inputs_HMI".SUSPENSÃO_CICLO_PRENSA )
      wire#w4
      S_Coil( "Etapas_Grafcet_1".SUSPENSÃO_CICLO )
   END_RUNG
   RUNG wire#w1
      Contact( "Inputs_HMI".MODO_2 )
      wire#w3
      Contact( "TM2".Q )
   END_RUNG wire#w2
   RUNG wire#w3
      Contact( "PH301_CONT_PH" )
   END_RUNG wire#w2
   RUNG wire#w4
      R_Coil( "Etapas_Grafcet_1".ETAPA_6 )
   END_RUNG
   // the same network as SCL:
   IF "Etapas_Grafcet_1".ETAPA_6 AND ((NOT "Inputs_HMI".MODO_2 AND "PH301_CONT_PH" AND "TM2".Q) OR ("Inputs_HMI".MODO_2 AND ("TM2".Q OR "PH301_CONT_PH"))) AND "Inputs_HMI".SUSPENSÃO_CICLO_PRENSA THEN
       "Etapas_Grafcet_1".SUSPENSÃO_CICLO := TRUE;
       "Etapas_Grafcet_1".ETAPA_6 := FALSE;
   END_IF;
END_REGION

REGION Network 14: Reset Suspensão Ciclo
   RUNG wire#powerrail
      I_Contact( "Inputs_HMI".SUSPENSÃO_CICLO_PRENSA )
      R_Coil( "Etapas_Grafcet_1".SUSPENSÃO_CICLO )
   END_RUNG
   // the same network as SCL:
   IF NOT "Inputs_HMI".SUSPENSÃO_CICLO_PRENSA THEN "Etapas_Grafcet_1".SUSPENSÃO_CICLO := FALSE; END_IF;
END_REGION

REGION Network 15: Tempo do agitador MX201
   RUNG wire#powerrail
      Contact( "Etapas_Grafcet_1".ETAPA_4 )
      Contact( "Inputs_HMI".MAN_AUTO )
      Contact( "BOT_EMERGÊNCIA" )
      { S7_Templates := "time_type := Time" } "TM1".TON(pt := "Inputs_HMI".TEMP_REDUÇÃO, et =>)
   END_RUNG
   // the same network as SCL:
   "TM1".TON(IN := "Etapas_Grafcet_1".ETAPA_4 AND "Inputs_HMI".MAN_AUTO AND "BOT_EMERGÊNCIA",
             PT := "Inputs_HMI".TEMP_REDUÇÃO);
END_REGION

REGION Network 16: Tempo do agitador MX301
   RUNG wire#powerrail
      Contact( "Etapas_Grafcet_1".ETAPA_6 )
      Contact( "Inputs_HMI".MAN_AUTO )
      Contact( "BOT_EMERGÊNCIA" )
      { S7_Templates := "time_type := Time" } "TM2".TON(pt := "Inputs_HMI".TEMP_PRECIPITAÇÃO, et =>)
   END_RUNG
   // the same network as SCL:
   "TM2".TON(IN := "Etapas_Grafcet_1".ETAPA_6 AND "Inputs_HMI".MAN_AUTO AND "BOT_EMERGÊNCIA",
             PT := "Inputs_HMI".TEMP_PRECIPITAÇÃO);
END_REGION

REGION Network 17: Tempo de pré-alarme
   RUNG wire#powerrail
      Contact( "Etapas_Grafcet_1".ETAPA_8 )
      { S7_Templates := "time_type := Time" } "TM3".TON(pt := "Inputs_HMI".TEMP_ALARME, et =>)
   END_RUNG
   // the same network as SCL:
   "TM3".TON(IN := "Etapas_Grafcet_1".ETAPA_8, PT := "Inputs_HMI".TEMP_ALARME);
END_REGION

REGION Network 18: LS101_SR_SET
   RUNG wire#powerrail
      Contact( "LSH101_TK01" )
      wire#w1
      S_Coil( "Info_Ciclo".LS101_SR )
   END_RUNG
   RUNG wire#powerrail
      Contact( "Inputs_HMI".MAN_AUTO )
      Contact( "Inputs_HMI".START_CICLO )
   END_RUNG wire#w1
   // the same network as SCL:
   IF "LSH101_TK01" OR ("Inputs_HMI".MAN_AUTO AND "Inputs_HMI".START_CICLO) THEN
       "Info_Ciclo".LS101_SR := TRUE;
   END_IF;
END_REGION

REGION Network 19: LS101_SR_RESET
   RUNG wire#powerrail
      I_Contact( "LSL101_TK01" )
      R_Coil( "Info_Ciclo".LS101_SR )
   END_RUNG
   // the same network as SCL:
   IF NOT "LSL101_TK01" THEN "Info_Ciclo".LS101_SR := FALSE; END_IF;
END_REGION
END_FUNCTION

FUNCTION "Saídas" : Void   // FC2, LAD
{ S7_Optimized_Access := 'TRUE' }
VERSION : 0.1
// stored: AutoNumber true, IsIECCheckEnabled false, SetENOAutomatically false, UDAEnableTagReadback false
   VAR_TEMP   // added for the SCL form of the ladder/FBD networks
      _w1 : Bool;
   END_VAR
BEGIN

REGION Network 1: bomba de alimentação ao processo BS001A
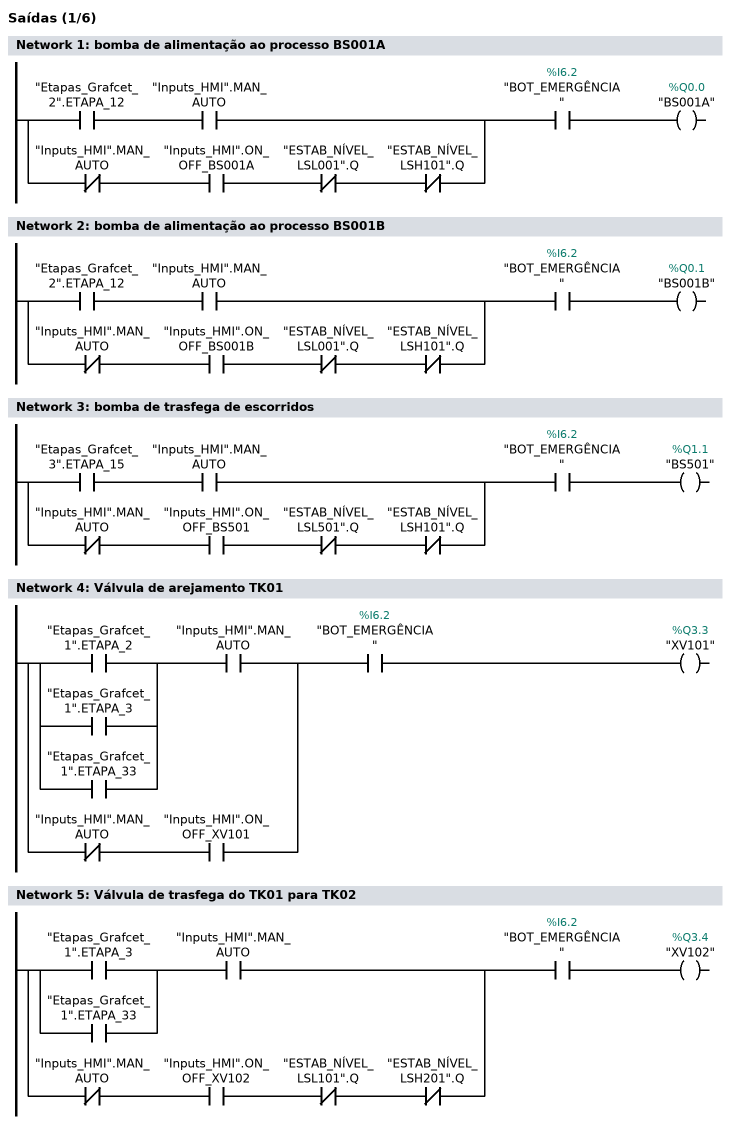
   RUNG wire#powerrail
      Contact( "Etapas_Grafcet_2".ETAPA_12 )
      Contact( "Inputs_HMI".MAN_AUTO )
      wire#w1
      Contact( "BOT_EMERGÊNCIA" )
      Coil( "BS001A" )
   END_RUNG
   RUNG wire#powerrail
      I_Contact( "Inputs_HMI".MAN_AUTO )
      Contact( "Inputs_HMI".ON_OFF_BS001A )
      I_Contact( "ESTAB_NÍVEL_LSL001".Q )
      I_Contact( "ESTAB_NÍVEL_LSH101".Q )
   END_RUNG wire#w1
   // the same network as SCL:
   "BS001A" := (("Etapas_Grafcet_2".ETAPA_12 AND "Inputs_HMI".MAN_AUTO) OR (NOT "Inputs_HMI".MAN_AUTO AND "Inputs_HMI".ON_OFF_BS001A AND NOT "ESTAB_NÍVEL_LSL001".Q AND NOT "ESTAB_NÍVEL_LSH101".Q)) AND "BOT_EMERGÊNCIA";
END_REGION

REGION Network 2: bomba de alimentação ao processo BS001B
   RUNG wire#powerrail
      Contact( "Etapas_Grafcet_2".ETAPA_12 )
      Contact( "Inputs_HMI".MAN_AUTO )
      wire#w1
      Contact( "BOT_EMERGÊNCIA" )
      Coil( "BS001B" )
   END_RUNG
   RUNG wire#powerrail
      I_Contact( "Inputs_HMI".MAN_AUTO )
      Contact( "Inputs_HMI".ON_OFF_BS001B )
      I_Contact( "ESTAB_NÍVEL_LSL001".Q )
      I_Contact( "ESTAB_NÍVEL_LSH101".Q )
   END_RUNG wire#w1
   // the same network as SCL:
   "BS001B" := (("Etapas_Grafcet_2".ETAPA_12 AND "Inputs_HMI".MAN_AUTO) OR (NOT "Inputs_HMI".MAN_AUTO AND "Inputs_HMI".ON_OFF_BS001B AND NOT "ESTAB_NÍVEL_LSL001".Q AND NOT "ESTAB_NÍVEL_LSH101".Q)) AND "BOT_EMERGÊNCIA";
END_REGION

REGION Network 3: bomba de trasfega de escorridos
   RUNG wire#powerrail
      Contact( "Etapas_Grafcet_3".ETAPA_15 )
      Contact( "Inputs_HMI".MAN_AUTO )
      wire#w1
      Contact( "BOT_EMERGÊNCIA" )
      Coil( "BS501" )
   END_RUNG
   RUNG wire#powerrail
      I_Contact( "Inputs_HMI".MAN_AUTO )
      Contact( "Inputs_HMI".ON_OFF_BS501 )
      I_Contact( "ESTAB_NÍVEL_LSL501".Q )
      I_Contact( "ESTAB_NÍVEL_LSH101".Q )
   END_RUNG wire#w1
   // the same network as SCL:
   "BS501" := (("Etapas_Grafcet_3".ETAPA_15 AND "Inputs_HMI".MAN_AUTO) OR (NOT "Inputs_HMI".MAN_AUTO AND "Inputs_HMI".ON_OFF_BS501 AND NOT "ESTAB_NÍVEL_LSL501".Q AND NOT "ESTAB_NÍVEL_LSH101".Q)) AND "BOT_EMERGÊNCIA";
END_REGION

REGION Network 4: Válvula de arejamento TK01
   RUNG wire#powerrail
      Contact( "Etapas_Grafcet_1".ETAPA_2 )
      wire#w1
      Contact( "Inputs_HMI".MAN_AUTO )
      wire#w2
      Contact( "BOT_EMERGÊNCIA" )
      Coil( "XV101" )
   END_RUNG
   RUNG wire#powerrail
      Contact( "Etapas_Grafcet_1".ETAPA_3 )
   END_RUNG wire#w1
   RUNG wire#powerrail
      Contact( "Etapas_Grafcet_1".ETAPA_33 )
   END_RUNG wire#w1
   RUNG wire#powerrail
      I_Contact( "Inputs_HMI".MAN_AUTO )
      Contact( "Inputs_HMI".ON_OFF_XV101 )
   END_RUNG wire#w2
   // the same network as SCL:
   "XV101" := ((("Etapas_Grafcet_1".ETAPA_2 OR "Etapas_Grafcet_1".ETAPA_3 OR "Etapas_Grafcet_1".ETAPA_33) AND "Inputs_HMI".MAN_AUTO) OR (NOT "Inputs_HMI".MAN_AUTO AND "Inputs_HMI".ON_OFF_XV101)) AND "BOT_EMERGÊNCIA";
END_REGION

REGION Network 5: Válvula de trasfega do TK01 para TK02
   RUNG wire#powerrail
      Contact( "Etapas_Grafcet_1".ETAPA_3 )
      wire#w1
      Contact( "Inputs_HMI".MAN_AUTO )
      wire#w2
      Contact( "BOT_EMERGÊNCIA" )
      Coil( "XV102" )
   END_RUNG
   RUNG wire#powerrail
      Contact( "Etapas_Grafcet_1".ETAPA_33 )
   END_RUNG wire#w1
   RUNG wire#powerrail
      I_Contact( "Inputs_HMI".MAN_AUTO )
      Contact( "Inputs_HMI".ON_OFF_XV102 )
      I_Contact( "ESTAB_NÍVEL_LSL101".Q )
      I_Contact( "ESTAB_NÍVEL_LSH201".Q )
   END_RUNG wire#w2
   // the same network as SCL:
   "XV102" := ((("Etapas_Grafcet_1".ETAPA_3 OR "Etapas_Grafcet_1".ETAPA_33) AND "Inputs_HMI".MAN_AUTO) OR (NOT "Inputs_HMI".MAN_AUTO AND "Inputs_HMI".ON_OFF_XV102 AND NOT "ESTAB_NÍVEL_LSL101".Q AND NOT "ESTAB_NÍVEL_LSH201".Q)) AND "BOT_EMERGÊNCIA";
END_REGION

REGION Network 6: Agitador MX201
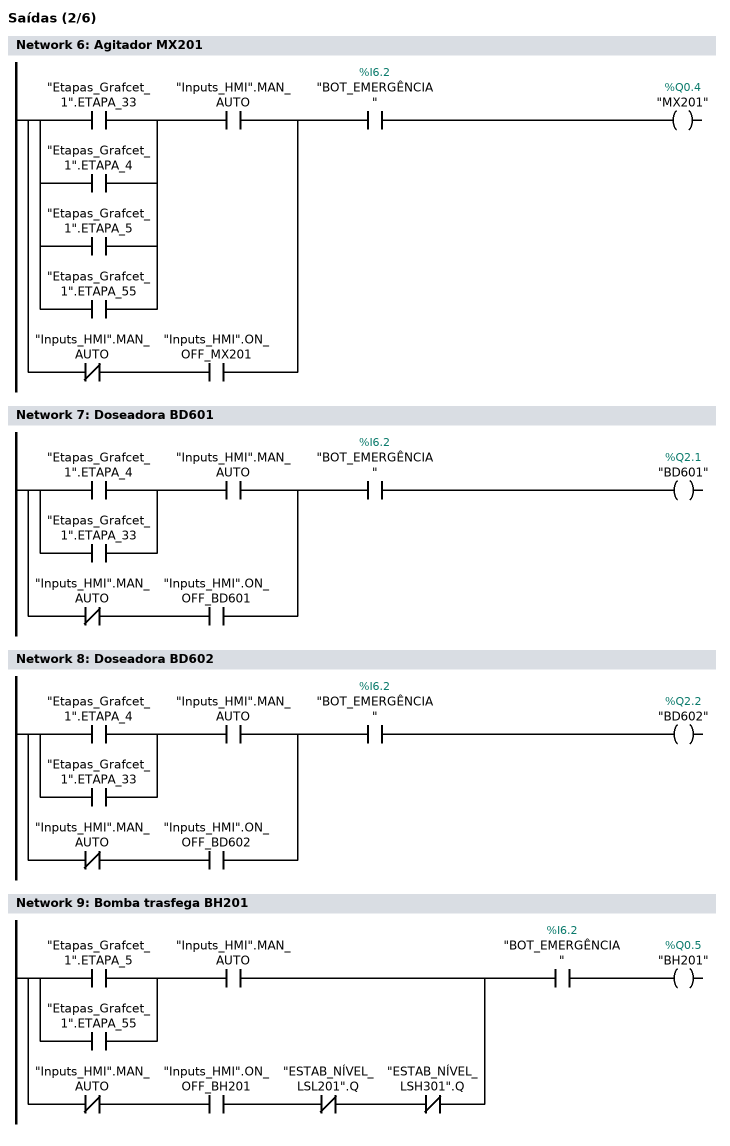
   RUNG wire#powerrail
      Contact( "Etapas_Grafcet_1".ETAPA_33 )
      wire#w1
      Contact( "Inputs_HMI".MAN_AUTO )
      wire#w2
      Contact( "BOT_EMERGÊNCIA" )
      Coil( "MX201" )
   END_RUNG
   RUNG wire#powerrail
      Contact( "Etapas_Grafcet_1".ETAPA_4 )
   END_RUNG wire#w1
   RUNG wire#powerrail
      Contact( "Etapas_Grafcet_1".ETAPA_5 )
   END_RUNG wire#w1
   RUNG wire#powerrail
      Contact( "Etapas_Grafcet_1".ETAPA_55 )
   END_RUNG wire#w1
   RUNG wire#powerrail
      I_Contact( "Inputs_HMI".MAN_AUTO )
      Contact( "Inputs_HMI".ON_OFF_MX201 )
   END_RUNG wire#w2
   // the same network as SCL:
   "MX201" := ((("Etapas_Grafcet_1".ETAPA_33 OR "Etapas_Grafcet_1".ETAPA_4 OR "Etapas_Grafcet_1".ETAPA_5 OR "Etapas_Grafcet_1".ETAPA_55) AND "Inputs_HMI".MAN_AUTO) OR (NOT "Inputs_HMI".MAN_AUTO AND "Inputs_HMI".ON_OFF_MX201)) AND "BOT_EMERGÊNCIA";
END_REGION

REGION Network 7: Doseadora BD601
   RUNG wire#powerrail
      Contact( "Etapas_Grafcet_1".ETAPA_4 )
      wire#w1
      Contact( "Inputs_HMI".MAN_AUTO )
      wire#w2
      Contact( "BOT_EMERGÊNCIA" )
      Coil( "BD601" )
   END_RUNG
   RUNG wire#powerrail
      Contact( "Etapas_Grafcet_1".ETAPA_33 )
   END_RUNG wire#w1
   RUNG wire#powerrail
      I_Contact( "Inputs_HMI".MAN_AUTO )
      Contact( "Inputs_HMI".ON_OFF_BD601 )
   END_RUNG wire#w2
   // the same network as SCL:
   "BD601" := ((("Etapas_Grafcet_1".ETAPA_4 OR "Etapas_Grafcet_1".ETAPA_33) AND "Inputs_HMI".MAN_AUTO) OR (NOT "Inputs_HMI".MAN_AUTO AND "Inputs_HMI".ON_OFF_BD601)) AND "BOT_EMERGÊNCIA";
END_REGION

REGION Network 8: Doseadora BD602
   RUNG wire#powerrail
      Contact( "Etapas_Grafcet_1".ETAPA_4 )
      wire#w1
      Contact( "Inputs_HMI".MAN_AUTO )
      wire#w2
      Contact( "BOT_EMERGÊNCIA" )
      Coil( "BD602" )
   END_RUNG
   RUNG wire#powerrail
      Contact( "Etapas_Grafcet_1".ETAPA_33 )
   END_RUNG wire#w1
   RUNG wire#powerrail
      I_Contact( "Inputs_HMI".MAN_AUTO )
      Contact( "Inputs_HMI".ON_OFF_BD602 )
   END_RUNG wire#w2
   // the same network as SCL:
   "BD602" := ((("Etapas_Grafcet_1".ETAPA_4 OR "Etapas_Grafcet_1".ETAPA_33) AND "Inputs_HMI".MAN_AUTO) OR (NOT "Inputs_HMI".MAN_AUTO AND "Inputs_HMI".ON_OFF_BD602)) AND "BOT_EMERGÊNCIA";
END_REGION

REGION Network 9: Bomba trasfega BH201
   RUNG wire#powerrail
      Contact( "Etapas_Grafcet_1".ETAPA_5 )
      wire#w1
      Contact( "Inputs_HMI".MAN_AUTO )
      wire#w2
      Contact( "BOT_EMERGÊNCIA" )
      Coil( "BH201" )
   END_RUNG
   RUNG wire#powerrail
      Contact( "Etapas_Grafcet_1".ETAPA_55 )
   END_RUNG wire#w1
   RUNG wire#powerrail
      I_Contact( "Inputs_HMI".MAN_AUTO )
      Contact( "Inputs_HMI".ON_OFF_BH201 )
      I_Contact( "ESTAB_NÍVEL_LSL201".Q )
      I_Contact( "ESTAB_NÍVEL_LSH301".Q )
   END_RUNG wire#w2
   // the same network as SCL:
   "BH201" := ((("Etapas_Grafcet_1".ETAPA_5 OR "Etapas_Grafcet_1".ETAPA_55) AND "Inputs_HMI".MAN_AUTO) OR (NOT "Inputs_HMI".MAN_AUTO AND "Inputs_HMI".ON_OFF_BH201 AND NOT "ESTAB_NÍVEL_LSL201".Q AND NOT "ESTAB_NÍVEL_LSH301".Q)) AND "BOT_EMERGÊNCIA";
END_REGION

REGION Network 10: Agitador MX301
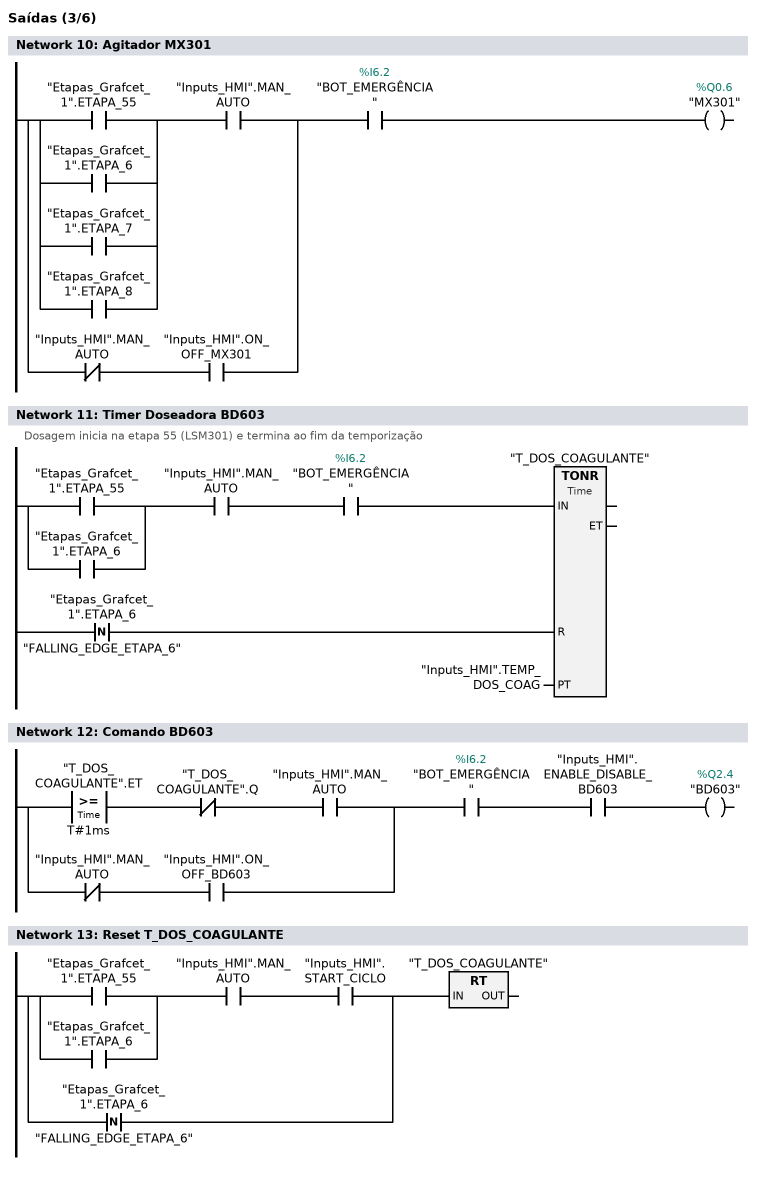
   RUNG wire#powerrail
      Contact( "Etapas_Grafcet_1".ETAPA_55 )
      wire#w1
      Contact( "Inputs_HMI".MAN_AUTO )
      wire#w2
      Contact( "BOT_EMERGÊNCIA" )
      Coil( "MX301" )
   END_RUNG
   RUNG wire#powerrail
      Contact( "Etapas_Grafcet_1".ETAPA_6 )
   END_RUNG wire#w1
   RUNG wire#powerrail
      Contact( "Etapas_Grafcet_1".ETAPA_7 )
   END_RUNG wire#w1
   RUNG wire#powerrail
      Contact( "Etapas_Grafcet_1".ETAPA_8 )
   END_RUNG wire#w1
   RUNG wire#powerrail
      I_Contact( "Inputs_HMI".MAN_AUTO )
      Contact( "Inputs_HMI".ON_OFF_MX301 )
   END_RUNG wire#w2
   // the same network as SCL:
   "MX301" := ((("Etapas_Grafcet_1".ETAPA_55 OR "Etapas_Grafcet_1".ETAPA_6 OR "Etapas_Grafcet_1".ETAPA_7 OR "Etapas_Grafcet_1".ETAPA_8) AND "Inputs_HMI".MAN_AUTO) OR (NOT "Inputs_HMI".MAN_AUTO AND "Inputs_HMI".ON_OFF_MX301)) AND "BOT_EMERGÊNCIA";
END_REGION

REGION Network 11: Timer Doseadora BD603
   // Dosagem inicia na etapa 55 (LSM301) e termina ao fim da temporização
   RUNG wire#powerrail
      Contact( "Etapas_Grafcet_1".ETAPA_55 )
      wire#w1
      Contact( "Inputs_HMI".MAN_AUTO )
      Contact( "BOT_EMERGÊNCIA" )
      { S7_Templates := "time_type := Time" } "T_DOS_COAGULANTE".TONR(r := wire#w2, pt := "Inputs_HMI".TEMP_DOS_COAG, et =>)
   END_RUNG
   RUNG wire#powerrail
      Contact( "Etapas_Grafcet_1".ETAPA_6 )
   END_RUNG wire#w1
   RUNG wire#powerrail
      N_Contact(operand := "Etapas_Grafcet_1".ETAPA_6, bit := "FALLING_EDGE_ETAPA_6")
   END_RUNG wire#w2
   // the same network as SCL:
   #_w1 := NOT "Etapas_Grafcet_1".ETAPA_6 AND "FALLING_EDGE_ETAPA_6";   // falling edge of "Etapas_Grafcet_1".ETAPA_6
   "FALLING_EDGE_ETAPA_6" := "Etapas_Grafcet_1".ETAPA_6;
   "T_DOS_COAGULANTE".TONR(IN := ("Etapas_Grafcet_1".ETAPA_55 OR "Etapas_Grafcet_1".ETAPA_6) AND "Inputs_HMI".MAN_AUTO AND "BOT_EMERGÊNCIA",
                           R := #_w1,
                           PT := "Inputs_HMI".TEMP_DOS_COAG);
END_REGION

REGION Network 12: Comando BD603
   RUNG wire#powerrail
      { S7_Templates := "SrcType := Time" } GE_Contact(in1 := "T_DOS_COAGULANTE".ET, in2 := T#1ms)
      I_Contact( "T_DOS_COAGULANTE".Q )
      Contact( "Inputs_HMI".MAN_AUTO )
      wire#w1
      Contact( "BOT_EMERGÊNCIA" )
      Contact( "Inputs_HMI".ENABLE_DISABLE_BD603 )
      Coil( "BD603" )
   END_RUNG
   RUNG wire#powerrail
      I_Contact( "Inputs_HMI".MAN_AUTO )
      Contact( "Inputs_HMI".ON_OFF_BD603 )
   END_RUNG wire#w1
   // the same network as SCL:
   "BD603" := ((("T_DOS_COAGULANTE".ET >= T#1ms) AND NOT "T_DOS_COAGULANTE".Q AND "Inputs_HMI".MAN_AUTO) OR (NOT "Inputs_HMI".MAN_AUTO AND "Inputs_HMI".ON_OFF_BD603)) AND "BOT_EMERGÊNCIA" AND "Inputs_HMI".ENABLE_DISABLE_BD603;
END_REGION

REGION Network 13: Reset T_DOS_COAGULANTE
   RUNG wire#powerrail
      Contact( "Etapas_Grafcet_1".ETAPA_55 )
      wire#w1
      Contact( "Inputs_HMI".MAN_AUTO )
      Contact( "Inputs_HMI".START_CICLO )
      wire#w2
      RT_Coil( "T_DOS_COAGULANTE" )
   END_RUNG
   RUNG wire#powerrail
      Contact( "Etapas_Grafcet_1".ETAPA_6 )
   END_RUNG wire#w1
   RUNG wire#powerrail
      N_Contact(operand := "Etapas_Grafcet_1".ETAPA_6, bit := "FALLING_EDGE_ETAPA_6")
   END_RUNG wire#w2
   // the same network as SCL:
   #_w1 := NOT "Etapas_Grafcet_1".ETAPA_6 AND "FALLING_EDGE_ETAPA_6";   // falling edge of "Etapas_Grafcet_1".ETAPA_6
   "FALLING_EDGE_ETAPA_6" := "Etapas_Grafcet_1".ETAPA_6;
   IF (("Etapas_Grafcet_1".ETAPA_55 OR "Etapas_Grafcet_1".ETAPA_6) AND "Inputs_HMI".MAN_AUTO AND "Inputs_HMI".START_CICLO) OR #_w1 THEN
       RESET_TIMER("T_DOS_COAGULANTE");
   END_IF;
END_REGION

REGION Network 14: Doseadora BD604
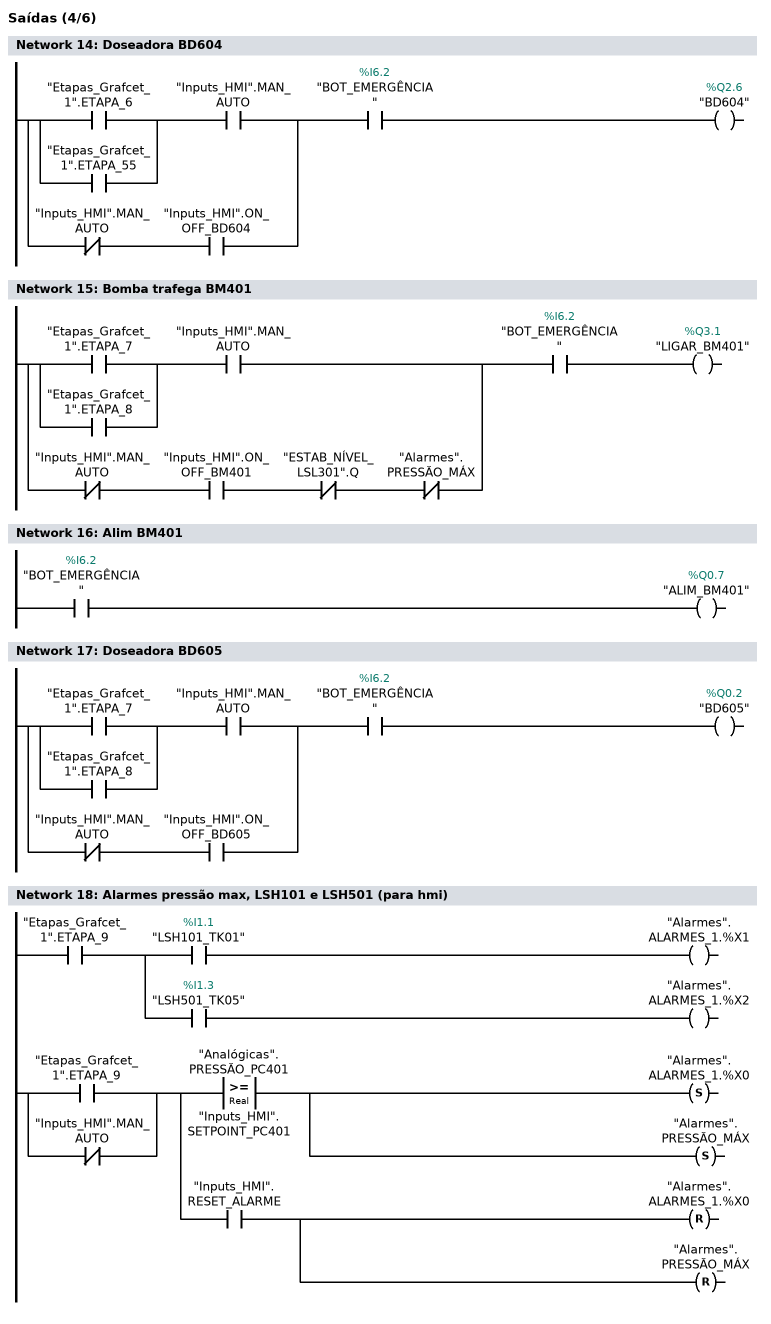
   RUNG wire#powerrail
      Contact( "Etapas_Grafcet_1".ETAPA_6 )
      wire#w1
      Contact( "Inputs_HMI".MAN_AUTO )
      wire#w2
      Contact( "BOT_EMERGÊNCIA" )
      Coil( "BD604" )
   END_RUNG
   RUNG wire#powerrail
      Contact( "Etapas_Grafcet_1".ETAPA_55 )
   END_RUNG wire#w1
   RUNG wire#powerrail
      I_Contact( "Inputs_HMI".MAN_AUTO )
      Contact( "Inputs_HMI".ON_OFF_BD604 )
   END_RUNG wire#w2
   // the same network as SCL:
   "BD604" := ((("Etapas_Grafcet_1".ETAPA_6 OR "Etapas_Grafcet_1".ETAPA_55) AND "Inputs_HMI".MAN_AUTO) OR (NOT "Inputs_HMI".MAN_AUTO AND "Inputs_HMI".ON_OFF_BD604)) AND "BOT_EMERGÊNCIA";
END_REGION

REGION Network 15: Bomba trafega BM401
   RUNG wire#powerrail
      Contact( "Etapas_Grafcet_1".ETAPA_7 )
      wire#w1
      Contact( "Inputs_HMI".MAN_AUTO )
      wire#w2
      Contact( "BOT_EMERGÊNCIA" )
      Coil( "LIGAR_BM401" )
   END_RUNG
   RUNG wire#powerrail
      Contact( "Etapas_Grafcet_1".ETAPA_8 )
   END_RUNG wire#w1
   RUNG wire#powerrail
      I_Contact( "Inputs_HMI".MAN_AUTO )
      Contact( "Inputs_HMI".ON_OFF_BM401 )
      I_Contact( "ESTAB_NÍVEL_LSL301".Q )
      I_Contact( "Alarmes".PRESSÃO_MÁX )
   END_RUNG wire#w2
   // the same network as SCL:
   "LIGAR_BM401" := ((("Etapas_Grafcet_1".ETAPA_7 OR "Etapas_Grafcet_1".ETAPA_8) AND "Inputs_HMI".MAN_AUTO) OR (NOT "Inputs_HMI".MAN_AUTO AND "Inputs_HMI".ON_OFF_BM401 AND NOT "ESTAB_NÍVEL_LSL301".Q AND NOT "Alarmes".PRESSÃO_MÁX)) AND "BOT_EMERGÊNCIA";
END_REGION

REGION Network 16: Alim BM401
   RUNG wire#powerrail
      Contact( "BOT_EMERGÊNCIA" )
      Coil( "ALIM_BM401" )
   END_RUNG
   // the same network as SCL:
   "ALIM_BM401" := "BOT_EMERGÊNCIA";
END_REGION

REGION Network 17: Doseadora BD605
   RUNG wire#powerrail
      Contact( "Etapas_Grafcet_1".ETAPA_7 )
      wire#w1
      Contact( "Inputs_HMI".MAN_AUTO )
      wire#w2
      Contact( "BOT_EMERGÊNCIA" )
      Coil( "BD605" )
   END_RUNG
   RUNG wire#powerrail
      Contact( "Etapas_Grafcet_1".ETAPA_8 )
   END_RUNG wire#w1
   RUNG wire#powerrail
      I_Contact( "Inputs_HMI".MAN_AUTO )
      Contact( "Inputs_HMI".ON_OFF_BD605 )
   END_RUNG wire#w2
   // the same network as SCL:
   "BD605" := ((("Etapas_Grafcet_1".ETAPA_7 OR "Etapas_Grafcet_1".ETAPA_8) AND "Inputs_HMI".MAN_AUTO) OR (NOT "Inputs_HMI".MAN_AUTO AND "Inputs_HMI".ON_OFF_BD605)) AND "BOT_EMERGÊNCIA";
END_REGION

REGION Network 18: Alarmes pressão max, LSH101 e LSH501 (para hmi)
   RUNG wire#powerrail
      Contact( "Etapas_Grafcet_1".ETAPA_9 )
      wire#w1
      Contact( "LSH101_TK01" )
      Coil( "Alarmes".ALARMES_1.%X1 )
   END_RUNG
   RUNG wire#w1
      Contact( "LSH501_TK05" )
      Coil( "Alarmes".ALARMES_1.%X2 )
   END_RUNG
   RUNG wire#powerrail
      Contact( "Etapas_Grafcet_1".ETAPA_9 )
      wire#w2
      { S7_Templates := "SrcType := Real" } GE_Contact(in1 := "Analógicas".PRESSÃO_PC401, in2 := "Inputs_HMI".SETPOINT_PC401)
      wire#w3
      S_Coil( "Alarmes".ALARMES_1.%X0 )
   END_RUNG
   RUNG wire#powerrail
      I_Contact( "Inputs_HMI".MAN_AUTO )
   END_RUNG wire#w2
   RUNG wire#w3
      S_Coil( "Alarmes".PRESSÃO_MÁX )
   END_RUNG
   RUNG wire#w2
      Contact( "Inputs_HMI".RESET_ALARME )
      wire#w4
      R_Coil( "Alarmes".ALARMES_1.%X0 )
   END_RUNG
   RUNG wire#w4
      R_Coil( "Alarmes".PRESSÃO_MÁX )
   END_RUNG
   // the same network as SCL:
   "Alarmes".ALARMES_1.%X1 := "Etapas_Grafcet_1".ETAPA_9 AND "LSH101_TK01";
   "Alarmes".ALARMES_1.%X2 := "Etapas_Grafcet_1".ETAPA_9 AND "LSH501_TK05";
   #_w1 := "Etapas_Grafcet_1".ETAPA_9 OR NOT "Inputs_HMI".MAN_AUTO;
   IF #_w1 AND ("Analógicas".PRESSÃO_PC401 >= "Inputs_HMI".SETPOINT_PC401) THEN
       "Alarmes".ALARMES_1.%X0 := TRUE;
       "Alarmes".PRESSÃO_MÁX := TRUE;
   END_IF;
   IF #_w1 AND "Inputs_HMI".RESET_ALARME THEN
       "Alarmes".ALARMES_1.%X0 := FALSE;
       "Alarmes".PRESSÃO_MÁX := FALSE;
   END_IF;
END_REGION

REGION Network 19: Alarme (luminoso)
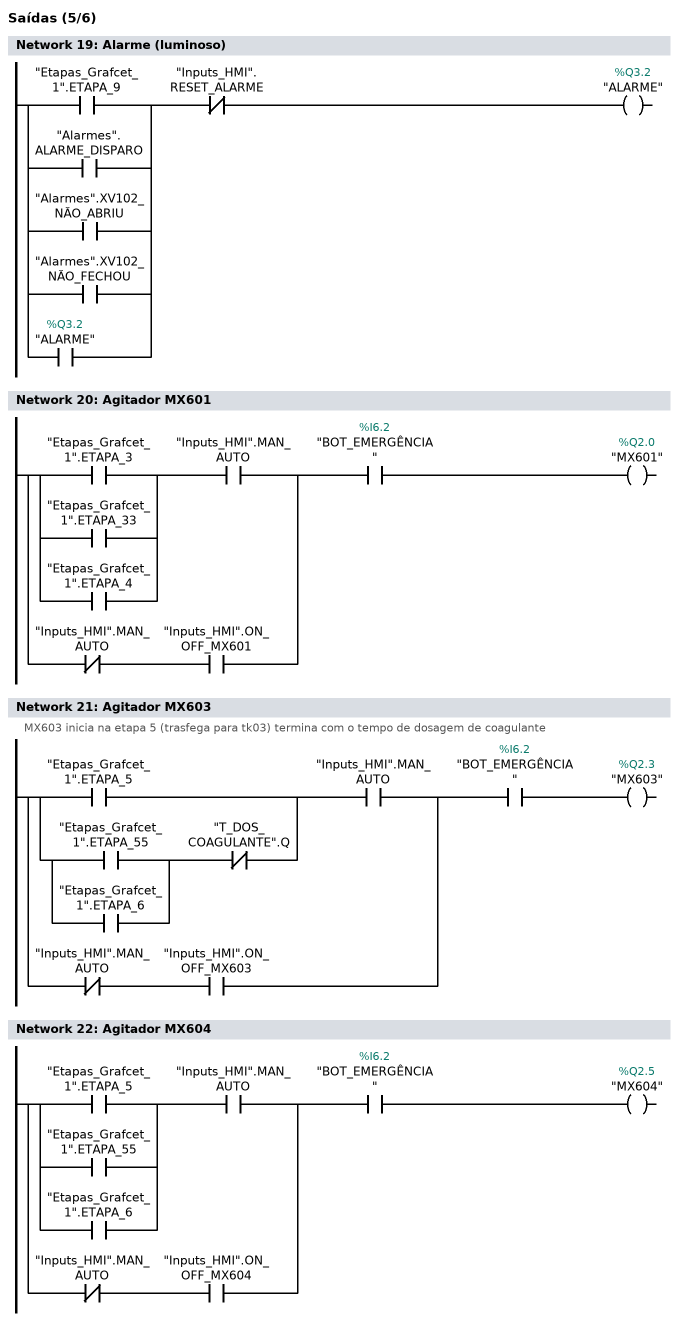
   RUNG wire#powerrail
      Contact( "Etapas_Grafcet_1".ETAPA_9 )
      wire#w1
      I_Contact( "Inputs_HMI".RESET_ALARME )
      Coil( "ALARME" )
   END_RUNG
   RUNG wire#powerrail
      Contact( "Alarmes".ALARME_DISPARO )
   END_RUNG wire#w1
   RUNG wire#powerrail
      Contact( "Alarmes".XV102_NÃO_ABRIU )
   END_RUNG wire#w1
   RUNG wire#powerrail
      Contact( "Alarmes".XV102_NÃO_FECHOU )
   END_RUNG wire#w1
   RUNG wire#powerrail
      Contact( "ALARME" )
   END_RUNG wire#w1
   // the same network as SCL:
   "ALARME" := ("Etapas_Grafcet_1".ETAPA_9 OR "Alarmes".ALARME_DISPARO OR "Alarmes".XV102_NÃO_ABRIU OR "Alarmes".XV102_NÃO_FECHOU OR "ALARME") AND NOT "Inputs_HMI".RESET_ALARME;
END_REGION

REGION Network 20: Agitador MX601
   RUNG wire#powerrail
      Contact( "Etapas_Grafcet_1".ETAPA_3 )
      wire#w1
      Contact( "Inputs_HMI".MAN_AUTO )
      wire#w2
      Contact( "BOT_EMERGÊNCIA" )
      Coil( "MX601" )
   END_RUNG
   RUNG wire#powerrail
      Contact( "Etapas_Grafcet_1".ETAPA_33 )
   END_RUNG wire#w1
   RUNG wire#powerrail
      Contact( "Etapas_Grafcet_1".ETAPA_4 )
   END_RUNG wire#w1
   RUNG wire#powerrail
      I_Contact( "Inputs_HMI".MAN_AUTO )
      Contact( "Inputs_HMI".ON_OFF_MX601 )
   END_RUNG wire#w2
   // the same network as SCL:
   "MX601" := ((("Etapas_Grafcet_1".ETAPA_3 OR "Etapas_Grafcet_1".ETAPA_33 OR "Etapas_Grafcet_1".ETAPA_4) AND "Inputs_HMI".MAN_AUTO) OR (NOT "Inputs_HMI".MAN_AUTO AND "Inputs_HMI".ON_OFF_MX601)) AND "BOT_EMERGÊNCIA";
END_REGION

REGION Network 21: Agitador MX603
   // MX603 inicia na etapa 5 (trasfega para tk03) termina com o tempo de dosagem de coagulante
   RUNG wire#powerrail
      Contact( "Etapas_Grafcet_1".ETAPA_5 )
      wire#w1
      Contact( "Inputs_HMI".MAN_AUTO )
      wire#w3
      Contact( "BOT_EMERGÊNCIA" )
      Coil( "MX603" )
   END_RUNG
   RUNG wire#powerrail
      Contact( "Etapas_Grafcet_1".ETAPA_55 )
      wire#w2
      I_Contact( "T_DOS_COAGULANTE".Q )
   END_RUNG wire#w1
   RUNG wire#powerrail
      Contact( "Etapas_Grafcet_1".ETAPA_6 )
   END_RUNG wire#w2
   RUNG wire#powerrail
      I_Contact( "Inputs_HMI".MAN_AUTO )
      Contact( "Inputs_HMI".ON_OFF_MX603 )
   END_RUNG wire#w3
   // the same network as SCL:
   "MX603" := ((("Etapas_Grafcet_1".ETAPA_5 OR (("Etapas_Grafcet_1".ETAPA_55 OR "Etapas_Grafcet_1".ETAPA_6) AND NOT "T_DOS_COAGULANTE".Q)) AND "Inputs_HMI".MAN_AUTO) OR (NOT "Inputs_HMI".MAN_AUTO AND "Inputs_HMI".ON_OFF_MX603)) AND "BOT_EMERGÊNCIA";
END_REGION

REGION Network 22: Agitador MX604
   RUNG wire#powerrail
      Contact( "Etapas_Grafcet_1".ETAPA_5 )
      wire#w1
      Contact( "Inputs_HMI".MAN_AUTO )
      wire#w2
      Contact( "BOT_EMERGÊNCIA" )
      Coil( "MX604" )
   END_RUNG
   RUNG wire#powerrail
      Contact( "Etapas_Grafcet_1".ETAPA_55 )
   END_RUNG wire#w1
   RUNG wire#powerrail
      Contact( "Etapas_Grafcet_1".ETAPA_6 )
   END_RUNG wire#w1
   RUNG wire#powerrail
      I_Contact( "Inputs_HMI".MAN_AUTO )
      Contact( "Inputs_HMI".ON_OFF_MX604 )
   END_RUNG wire#w2
   // the same network as SCL:
   "MX604" := ((("Etapas_Grafcet_1".ETAPA_5 OR "Etapas_Grafcet_1".ETAPA_55 OR "Etapas_Grafcet_1".ETAPA_6) AND "Inputs_HMI".MAN_AUTO) OR (NOT "Inputs_HMI".MAN_AUTO AND "Inputs_HMI".ON_OFF_MX604)) AND "BOT_EMERGÊNCIA";
END_REGION

REGION Network 23: Agitador MX605
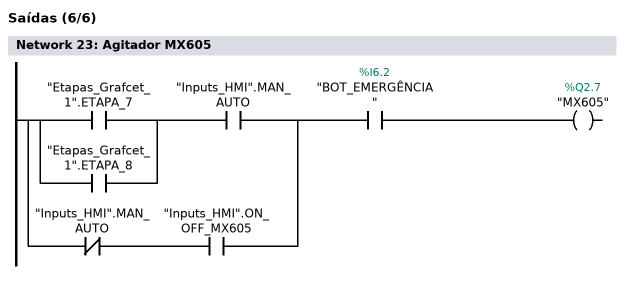
   RUNG wire#powerrail
      Contact( "Etapas_Grafcet_1".ETAPA_7 )
      wire#w1
      Contact( "Inputs_HMI".MAN_AUTO )
      wire#w2
      Contact( "BOT_EMERGÊNCIA" )
      Coil( "MX605" )
   END_RUNG
   RUNG wire#powerrail
      Contact( "Etapas_Grafcet_1".ETAPA_8 )
   END_RUNG wire#w1
   RUNG wire#powerrail
      I_Contact( "Inputs_HMI".MAN_AUTO )
      Contact( "Inputs_HMI".ON_OFF_MX605 )
   END_RUNG wire#w2
   // the same network as SCL:
   "MX605" := ((("Etapas_Grafcet_1".ETAPA_7 OR "Etapas_Grafcet_1".ETAPA_8) AND "Inputs_HMI".MAN_AUTO) OR (NOT "Inputs_HMI".MAN_AUTO AND "Inputs_HMI".ON_OFF_MX605)) AND "BOT_EMERGÊNCIA";
END_REGION
END_FUNCTION

FUNCTION "Níveis_TK02" : Void   // FC5, LAD
{ S7_Optimized_Access := 'TRUE' }
VERSION : 0.1
// stored: AutoNumber true, IsIECCheckEnabled false, SetENOAutomatically false, UDAEnableTagReadback false
BEGIN

REGION Network 1
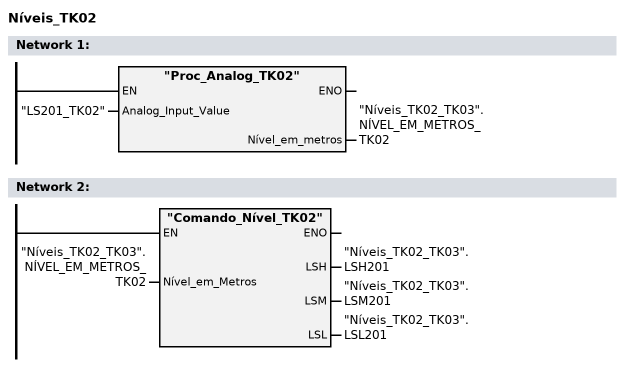
   RUNG wire#powerrail
      "Proc_Analog_TK02"(Analog_Input_Value := "LS201_TK02", Nível_em_metros => "Níveis_TK02_TK03".NÍVEL_EM_METROS_TK02)
   END_RUNG
   // the same network as SCL:
   "Proc_Analog_TK02"(Analog_Input_Value := "LS201_TK02",
                      Nível_em_metros => "Níveis_TK02_TK03".NÍVEL_EM_METROS_TK02);
END_REGION

REGION Network 2
   RUNG wire#powerrail
      "Comando_Nível_TK02"(Nível_em_Metros := "Níveis_TK02_TK03".NÍVEL_EM_METROS_TK02, LSH => "Níveis_TK02_TK03".LSH201, LSM => "Níveis_TK02_TK03".LSM201, LSL => "Níveis_TK02_TK03".LSL201)
   END_RUNG
   // the same network as SCL:
   "Comando_Nível_TK02"(Nível_em_Metros := "Níveis_TK02_TK03".NÍVEL_EM_METROS_TK02,
                        LSH => "Níveis_TK02_TK03".LSH201,
                        LSM => "Níveis_TK02_TK03".LSM201,
                        LSL => "Níveis_TK02_TK03".LSL201);
END_REGION
END_FUNCTION

FUNCTION "Proc_Analog_TK02" : Void   // FC6, LAD
{ S7_Optimized_Access := 'TRUE' }
VERSION : 0.1
// stored: AutoNumber true, IsIECCheckEnabled false, SetENOAutomatically false, UDAEnableTagReadback false
   VAR_INPUT
      Analog_Input_Value : Int;
   END_VAR
   VAR_OUTPUT
      Nível_em_metros : Real;
   END_VAR
   VAR_TEMP
      "Nível_em_%" : Real;
   END_VAR
BEGIN

REGION Network 1
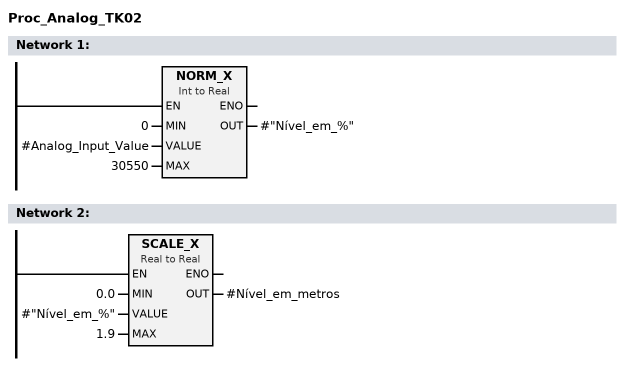
   RUNG wire#powerrail
      { S7_Templates := "[SrcType := Int, DestType := Real]"; S7_GenerateENO := "TRUE" } Normalize(min := 0, value := #Analog_Input_Value, max := 30550, out => #"Nível_em_%")
   END_RUNG
   // the same network as SCL:
   #"Nível_em_%" := NORM_X(MIN := 0, VALUE := #Analog_Input_Value, MAX := 30550);
END_REGION

REGION Network 2
   RUNG wire#powerrail
      { S7_Templates := "[SrcType := Real, DestType := Real]"; S7_GenerateENO := "TRUE" } Scale(min := 0.0, value := #"Nível_em_%", max := 1.9, out => #Nível_em_metros)
   END_RUNG
   // the same network as SCL:
   #Nível_em_metros := SCALE_X(MIN := 0.0, VALUE := #"Nível_em_%", MAX := 1.9);
END_REGION
END_FUNCTION

FUNCTION "Comando_Nível_TK02" : Void   // FC7, LAD
{ S7_Optimized_Access := 'TRUE' }
VERSION : 0.1
// stored: AutoNumber true, IsIECCheckEnabled false, SetENOAutomatically false, UDAEnableTagReadback false
   VAR_INPUT
      Nível_em_Metros : Real;
   END_VAR
   VAR_OUTPUT
      LSH : Bool;
      LSM : Bool;
      LSL : Bool;
   END_VAR
BEGIN

REGION Network 1
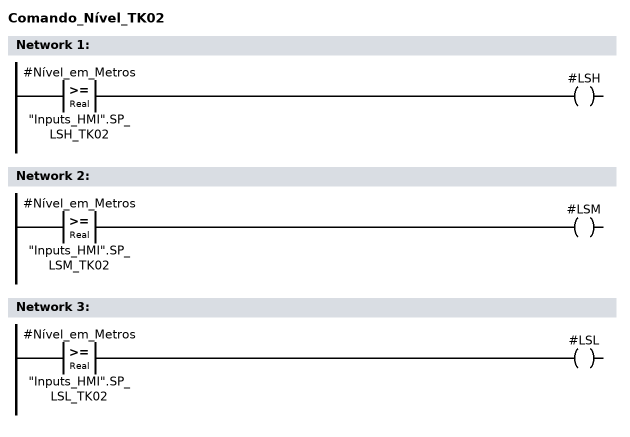
   RUNG wire#powerrail
      { S7_Templates := "SrcType := Real" } GE_Contact(in1 := #Nível_em_Metros, in2 := "Inputs_HMI".SP_LSH_TK02)
      Coil( #LSH )
   END_RUNG
   // the same network as SCL:
   #LSH := #Nível_em_Metros >= "Inputs_HMI".SP_LSH_TK02;
END_REGION

REGION Network 2
   RUNG wire#powerrail
      { S7_Templates := "SrcType := Real" } GE_Contact(in1 := #Nível_em_Metros, in2 := "Inputs_HMI".SP_LSM_TK02)
      Coil( #LSM )
   END_RUNG
   // the same network as SCL:
   #LSM := #Nível_em_Metros >= "Inputs_HMI".SP_LSM_TK02;
END_REGION

REGION Network 3
   RUNG wire#powerrail
      { S7_Templates := "SrcType := Real" } GE_Contact(in1 := #Nível_em_Metros, in2 := "Inputs_HMI".SP_LSL_TK02)
      Coil( #LSL )
   END_RUNG
   // the same network as SCL:
   #LSL := #Nível_em_Metros >= "Inputs_HMI".SP_LSL_TK02;
END_REGION
END_FUNCTION

FUNCTION "Níveis_TK03" : Void   // FC8, LAD
{ S7_Optimized_Access := 'TRUE' }
VERSION : 0.1
// stored: AutoNumber true, IsIECCheckEnabled false, SetENOAutomatically false, UDAEnableTagReadback false
BEGIN

REGION Network 1
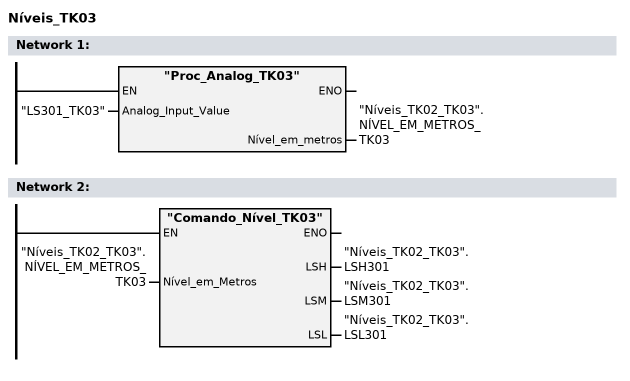
   RUNG wire#powerrail
      "Proc_Analog_TK03"(Analog_Input_Value := "LS301_TK03", Nível_em_metros => "Níveis_TK02_TK03".NÍVEL_EM_METROS_TK03)
   END_RUNG
   // the same network as SCL:
   "Proc_Analog_TK03"(Analog_Input_Value := "LS301_TK03",
                      Nível_em_metros => "Níveis_TK02_TK03".NÍVEL_EM_METROS_TK03);
END_REGION

REGION Network 2
   RUNG wire#powerrail
      "Comando_Nível_TK03"(Nível_em_Metros := "Níveis_TK02_TK03".NÍVEL_EM_METROS_TK03, LSH => "Níveis_TK02_TK03".LSH301, LSM => "Níveis_TK02_TK03".LSM301, LSL => "Níveis_TK02_TK03".LSL301)
   END_RUNG
   // the same network as SCL:
   "Comando_Nível_TK03"(Nível_em_Metros := "Níveis_TK02_TK03".NÍVEL_EM_METROS_TK03,
                        LSH => "Níveis_TK02_TK03".LSH301,
                        LSM => "Níveis_TK02_TK03".LSM301,
                        LSL => "Níveis_TK02_TK03".LSL301);
END_REGION
END_FUNCTION

FUNCTION "Proc_Analog_TK03" : Void   // FC9, LAD
{ S7_Optimized_Access := 'TRUE' }
VERSION : 0.1
// stored: AutoNumber true, IsIECCheckEnabled false, SetENOAutomatically false, UDAEnableTagReadback false
   VAR_INPUT
      Analog_Input_Value : Int;
   END_VAR
   VAR_OUTPUT
      Nível_em_metros : Real;
   END_VAR
   VAR_TEMP
      "Nível_em_%" : Real;
   END_VAR
BEGIN

REGION Network 1
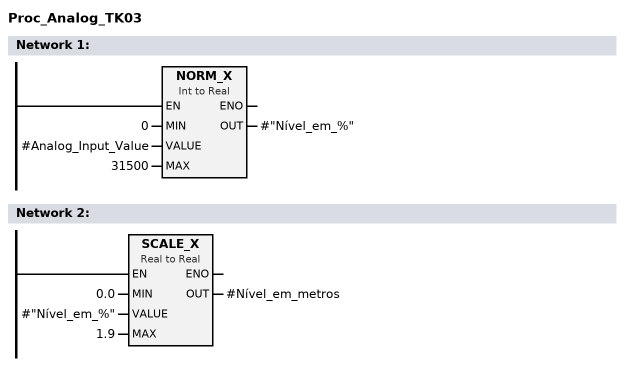
   RUNG wire#powerrail
      { S7_Templates := "[SrcType := Int, DestType := Real]"; S7_GenerateENO := "TRUE" } Normalize(min := 0, value := #Analog_Input_Value, max := 31500, out => #"Nível_em_%")
   END_RUNG
   // the same network as SCL:
   #"Nível_em_%" := NORM_X(MIN := 0, VALUE := #Analog_Input_Value, MAX := 31500);
END_REGION

REGION Network 2
   RUNG wire#powerrail
      { S7_Templates := "[SrcType := Real, DestType := Real]"; S7_GenerateENO := "TRUE" } Scale(min := 0.0, value := #"Nível_em_%", max := 1.9, out => #Nível_em_metros)
   END_RUNG
   // the same network as SCL:
   #Nível_em_metros := SCALE_X(MIN := 0.0, VALUE := #"Nível_em_%", MAX := 1.9);
END_REGION
END_FUNCTION

FUNCTION "Comando_Nível_TK03" : Void   // FC10, LAD
{ S7_Optimized_Access := 'TRUE' }
VERSION : 0.1
// stored: AutoNumber true, IsIECCheckEnabled false, SetENOAutomatically false, UDAEnableTagReadback false
   VAR_INPUT
      Nível_em_Metros : Real;
   END_VAR
   VAR_OUTPUT
      LSH : Bool;
      LSM : Bool;
      LSL : Bool;
   END_VAR
BEGIN

REGION Network 1
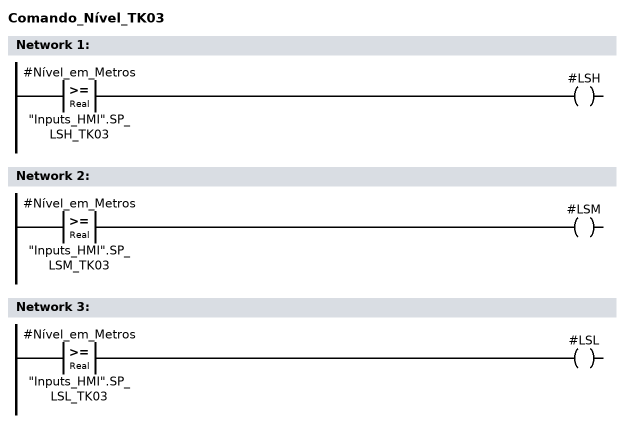
   RUNG wire#powerrail
      { S7_Templates := "SrcType := Real" } GE_Contact(in1 := #Nível_em_Metros, in2 := "Inputs_HMI".SP_LSH_TK03)
      Coil( #LSH )
   END_RUNG
   // the same network as SCL:
   #LSH := #Nível_em_Metros >= "Inputs_HMI".SP_LSH_TK03;
END_REGION

REGION Network 2
   RUNG wire#powerrail
      { S7_Templates := "SrcType := Real" } GE_Contact(in1 := #Nível_em_Metros, in2 := "Inputs_HMI".SP_LSM_TK03)
      Coil( #LSM )
   END_RUNG
   // the same network as SCL:
   #LSM := #Nível_em_Metros >= "Inputs_HMI".SP_LSM_TK03;
END_REGION

REGION Network 3
   RUNG wire#powerrail
      { S7_Templates := "SrcType := Real" } GE_Contact(in1 := #Nível_em_Metros, in2 := "Inputs_HMI".SP_LSL_TK03)
      Coil( #LSL )
   END_RUNG
   // the same network as SCL:
   #LSL := #Nível_em_Metros >= "Inputs_HMI".SP_LSL_TK03;
END_REGION
END_FUNCTION

FUNCTION "Medidor_Caudal_FQ301" : Void   // FC11, LAD
{ S7_Optimized_Access := 'TRUE' }
VERSION : 0.1
// stored: AutoNumber true, IsIECCheckEnabled false, SetENOAutomatically false, UDAEnableTagReadback false
BEGIN

REGION Network 1
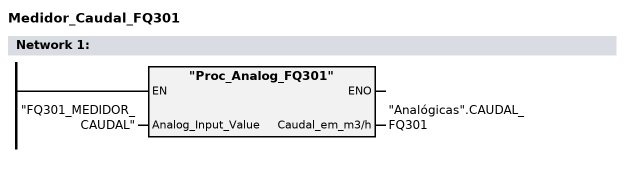
   RUNG wire#powerrail
      "Proc_Analog_FQ301"(Analog_Input_Value := "FQ301_MEDIDOR_CAUDAL", "Caudal_em_m3/h" => "Analógicas".CAUDAL_FQ301)
   END_RUNG
   // the same network as SCL:
   "Proc_Analog_FQ301"(Analog_Input_Value := "FQ301_MEDIDOR_CAUDAL",
                       "Caudal_em_m3/h" => "Analógicas".CAUDAL_FQ301);
END_REGION
END_FUNCTION

FUNCTION "Proc_Analog_FQ301" : Void   // FC12, LAD
{ S7_Optimized_Access := 'TRUE' }
VERSION : 0.1
// stored: AutoNumber true, IsIECCheckEnabled false, SetENOAutomatically false, UDAEnableTagReadback false
   VAR_INPUT
      Analog_Input_Value : Int;
   END_VAR
   VAR_OUTPUT
      "Caudal_em_m3/h" : Real;
   END_VAR
   VAR_TEMP
      "Caudal_em_%" : Real;
   END_VAR
BEGIN

REGION Network 1
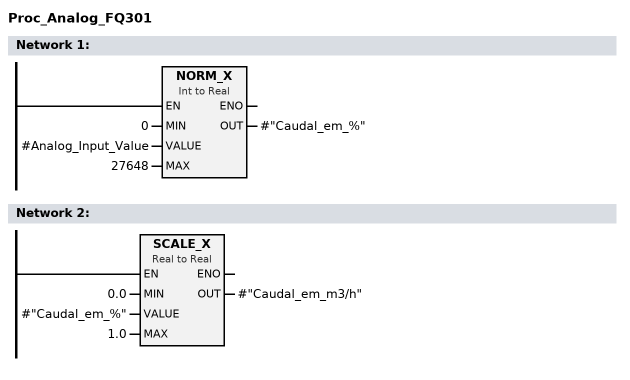
   RUNG wire#powerrail
      { S7_Templates := "[SrcType := Int, DestType := Real]"; S7_GenerateENO := "TRUE" } Normalize(min := 0, value := #Analog_Input_Value, max := 27648, out => #"Caudal_em_%")
   END_RUNG
   // the same network as SCL:
   #"Caudal_em_%" := NORM_X(MIN := 0, VALUE := #Analog_Input_Value, MAX := 27648);
END_REGION

REGION Network 2
   RUNG wire#powerrail
      { S7_Templates := "[SrcType := Real, DestType := Real]"; S7_GenerateENO := "TRUE" } Scale(min := 0.0, value := #"Caudal_em_%", max := 1.0, out => #"Caudal_em_m3/h")
   END_RUNG
   // the same network as SCL:
   #"Caudal_em_m3/h" := SCALE_X(MIN := 0.0, VALUE := #"Caudal_em_%", MAX := 1.0);
END_REGION
END_FUNCTION

FUNCTION "Sensor_Pressão_PC401" : Void   // FC13, LAD
{ S7_Optimized_Access := 'TRUE' }
VERSION : 0.1
// stored: AutoNumber true, IsIECCheckEnabled false, SetENOAutomatically false, UDAEnableTagReadback false
BEGIN

REGION Network 1
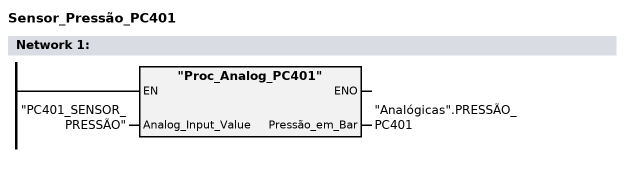
   RUNG wire#powerrail
      "Proc_Analog_PC401"(Analog_Input_Value := "PC401_SENSOR_PRESSÃO", Pressão_em_Bar => "Analógicas".PRESSÃO_PC401)
   END_RUNG
   // the same network as SCL:
   "Proc_Analog_PC401"(Analog_Input_Value := "PC401_SENSOR_PRESSÃO",
                       Pressão_em_Bar => "Analógicas".PRESSÃO_PC401);
END_REGION
END_FUNCTION

FUNCTION "Proc_Analog_PC401" : Void   // FC14, LAD
{ S7_Optimized_Access := 'TRUE' }
VERSION : 0.1
// stored: AutoNumber true, IsIECCheckEnabled false, SetENOAutomatically false, UDAEnableTagReadback false
   VAR_INPUT
      Analog_Input_Value : Int;
   END_VAR
   VAR_OUTPUT
      Pressão_em_Bar : Real;
   END_VAR
   VAR_TEMP
      "Pressão_em_%" : Real;
   END_VAR
BEGIN

REGION Network 1
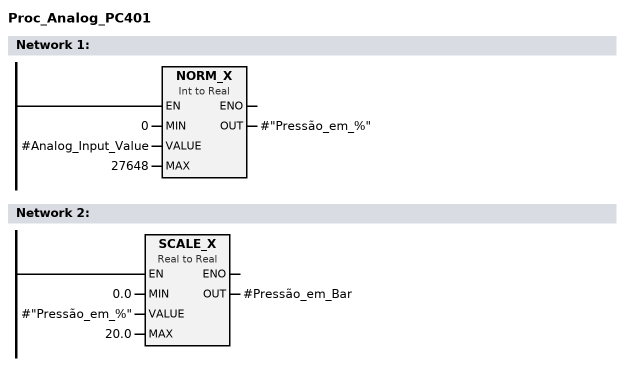
   RUNG wire#powerrail
      { S7_Templates := "[SrcType := Int, DestType := Real]"; S7_GenerateENO := "TRUE" } Normalize(min := 0, value := #Analog_Input_Value, max := 27648, out => #"Pressão_em_%")
   END_RUNG
   // the same network as SCL:
   #"Pressão_em_%" := NORM_X(MIN := 0, VALUE := #Analog_Input_Value, MAX := 27648);
END_REGION

REGION Network 2
   RUNG wire#powerrail
      { S7_Templates := "[SrcType := Real, DestType := Real]"; S7_GenerateENO := "TRUE" } Scale(min := 0.0, value := #"Pressão_em_%", max := 20.0, out => #Pressão_em_Bar)
   END_RUNG
   // the same network as SCL:
   #Pressão_em_Bar := SCALE_X(MIN := 0.0, VALUE := #"Pressão_em_%", MAX := 20.0);
END_REGION
END_FUNCTION

FUNCTION "Estados_HMI" : Void
{ S7_Optimized_Access := 'TRUE' }
VERSION : 0.1

BEGIN
	"Estados_HMI_DB".MX201 := "MX201_ON";
	"Estados_HMI_DB".MX601 := "MX601_ON";
	"Estados_HMI_DB".XV101 := "XV101_ABERTA";
	
	IF "XV102_ABERTA" = TRUE
	THEN
	    "Estados_HMI_DB".XV102 := TRUE;
	END_IF;
	
	IF "XV102_FECHADA" = TRUE
	THEN
	    "Estados_HMI_DB".XV102 := FALSE;
	END_IF;
	
	"Estados_HMI_DB".BD601 := "BD601_ON";
	"Estados_HMI_DB".BD602 := "BD602_ON";
	"Estados_HMI_DB".BH201 := "BH201_ON";
	"Estados_HMI_DB".PH201 := "PH201_CONT_PH";
	"Estados_HMI_DB".RH201 := "RH201_CONT_REDOX";
	"Estados_HMI_DB".MX603 := "MX603_ON";
	"Estados_HMI_DB".BD603 := "BD603_ON";
	"Estados_HMI_DB".MX301 := "MX301_ON";
	"Estados_HMI_DB".PH301 := "PH301_CONT_PH";
	"Estados_HMI_DB".BM401 := "BM401_ON";
	"Estados_HMI_DB".MX604 := "MX604_ON";
	"Estados_HMI_DB".BD604 := "BD604_ON";
	"Estados_HMI_DB".MX605 := "MX605_ON";
	"Estados_HMI_DB".BD605 := "BD605_ON";
	"Estados_HMI_DB".BS001A := "BS001A_ON";
	"Estados_HMI_DB".BS001B := "BS001B_ON";
	"Estados_HMI_DB".BS501 := "BS501_ON";
END_FUNCTION

FUNCTION "Encrav_Inputs_HMI" : Void
{ S7_Optimized_Access := 'TRUE' }
VERSION : 0.1

BEGIN
	IF "Inputs_HMI".MAN_AUTO = TRUE THEN
	    "Inputs_HMI".ON_OFF_MX201 := FALSE;
	    "Inputs_HMI".ON_OFF_MX301 := FALSE;
	    "Inputs_HMI".ON_OFF_MX601 := FALSE;
	    "Inputs_HMI".ON_OFF_MX603 := FALSE;
	    "Inputs_HMI".ON_OFF_MX604 := FALSE;
	    "Inputs_HMI".ON_OFF_MX605 := FALSE;
	    "Inputs_HMI".ON_OFF_BS001A := FALSE;
	    "Inputs_HMI".ON_OFF_BS001B := FALSE;
	    "Inputs_HMI".ON_OFF_BS501 := FALSE;
	    "Inputs_HMI".ON_OFF_BH201 := FALSE;
	    "Inputs_HMI".ON_OFF_BM401 := FALSE;
	    "Inputs_HMI".ON_OFF_BD601 := FALSE;
	    "Inputs_HMI".ON_OFF_BD602 := FALSE;
	    "Inputs_HMI".ON_OFF_BD603 := FALSE;
	    "Inputs_HMI".ON_OFF_BD604 := FALSE;
	    "Inputs_HMI".ON_OFF_BD605 := FALSE;
	    "Inputs_HMI".ON_OFF_XV101 := FALSE;
	    "Inputs_HMI".ON_OFF_XV102 := FALSE;
	END_IF;
END_FUNCTION

FUNCTION "Estado_Ciclo_HMI" : Void
{ S7_Optimized_Access := 'TRUE' }
VERSION : 0.1

BEGIN
	IF ("Etapas_Grafcet_1".ETAPA_1 = TRUE) OR ("Inputs_HMI".MAN_AUTO = FALSE) OR ("BOT_EMERGÊNCIA" = FALSE) THEN
	    "Info_Ciclo".ESTADO_CICLO := FALSE;
	ELSE
	    "Info_Ciclo".ESTADO_CICLO := TRUE;
	END_IF;
END_FUNCTION

FUNCTION "Alarmes_Disparos_1" : Void   // FC22, LAD
{ S7_Optimized_Access := 'TRUE' }
VERSION : 0.1
// stored: AutoNumber true, IsIECCheckEnabled false, SetENOAutomatically false, UDAEnableTagReadback false
   VAR_TEMP   // added for the SCL form of the ladder/FBD networks
      _w1 : Bool;
      _w2 : Bool;
      _w3 : Bool;
      _w4 : Bool;
      _w5 : Bool;
      _w6 : Bool;
      _w7 : Bool;
      _w8 : Bool;
      _w9 : Bool;
      _w10 : Bool;
      _w11 : Bool;
      _w12 : Bool;
      _w13 : Bool;
      _w14 : Bool;
      _w15 : Bool;
      _w16 : Bool;
      _w17 : Bool;
      _w18 : Bool;
      _w19 : Bool;
      _w20 : Bool;
      _w21 : Bool;
      _w22 : Bool;
   END_VAR
BEGIN

REGION Network 1: Ativa contacto de alarme disparos para alarme luminoso
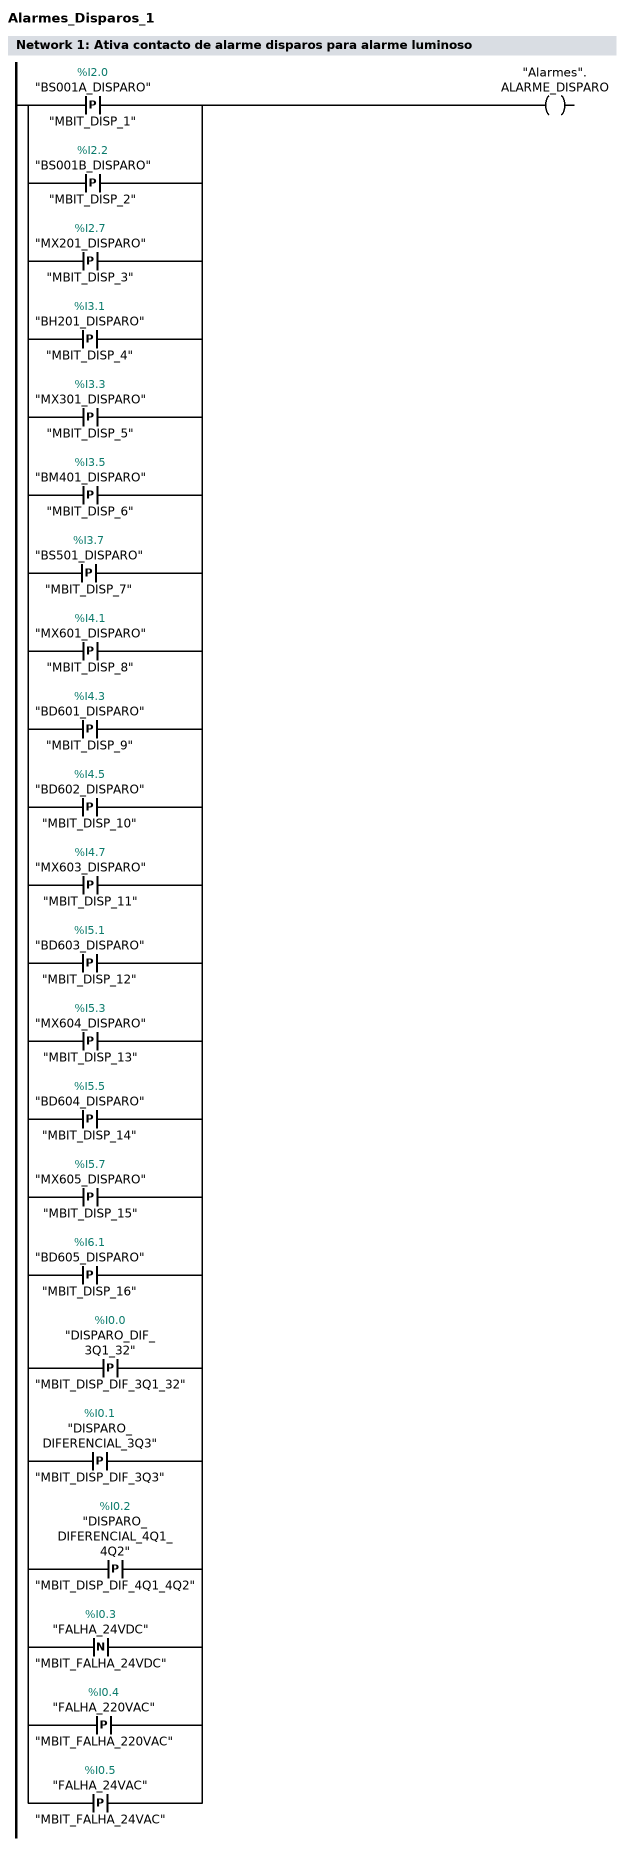
   RUNG wire#powerrail
      P_Contact(operand := "BS001A_DISPARO", bit := "MBIT_DISP_1")
      wire#w1
      Coil( "Alarmes".ALARME_DISPARO )
   END_RUNG
   RUNG wire#powerrail
      P_Contact(operand := "BS001B_DISPARO", bit := "MBIT_DISP_2")
   END_RUNG wire#w1
   RUNG wire#powerrail
      P_Contact(operand := "MX201_DISPARO", bit := "MBIT_DISP_3")
   END_RUNG wire#w1
   RUNG wire#powerrail
      P_Contact(operand := "BH201_DISPARO", bit := "MBIT_DISP_4")
   END_RUNG wire#w1
   RUNG wire#powerrail
      P_Contact(operand := "MX301_DISPARO", bit := "MBIT_DISP_5")
   END_RUNG wire#w1
   RUNG wire#powerrail
      P_Contact(operand := "BM401_DISPARO", bit := "MBIT_DISP_6")
   END_RUNG wire#w1
   RUNG wire#powerrail
      P_Contact(operand := "BS501_DISPARO", bit := "MBIT_DISP_7")
   END_RUNG wire#w1
   RUNG wire#powerrail
      P_Contact(operand := "MX601_DISPARO", bit := "MBIT_DISP_8")
   END_RUNG wire#w1
   RUNG wire#powerrail
      P_Contact(operand := "BD601_DISPARO", bit := "MBIT_DISP_9")
   END_RUNG wire#w1
   RUNG wire#powerrail
      P_Contact(operand := "BD602_DISPARO", bit := "MBIT_DISP_10")
   END_RUNG wire#w1
   RUNG wire#powerrail
      P_Contact(operand := "MX603_DISPARO", bit := "MBIT_DISP_11")
   END_RUNG wire#w1
   RUNG wire#powerrail
      P_Contact(operand := "BD603_DISPARO", bit := "MBIT_DISP_12")
   END_RUNG wire#w1
   RUNG wire#powerrail
      P_Contact(operand := "MX604_DISPARO", bit := "MBIT_DISP_13")
   END_RUNG wire#w1
   RUNG wire#powerrail
      P_Contact(operand := "BD604_DISPARO", bit := "MBIT_DISP_14")
   END_RUNG wire#w1
   RUNG wire#powerrail
      P_Contact(operand := "MX605_DISPARO", bit := "MBIT_DISP_15")
   END_RUNG wire#w1
   RUNG wire#powerrail
      P_Contact(operand := "BD605_DISPARO", bit := "MBIT_DISP_16")
   END_RUNG wire#w1
   RUNG wire#powerrail
      P_Contact(operand := "DISPARO_DIF_3Q1_32", bit := "MBIT_DISP_DIF_3Q1_32")
   END_RUNG wire#w1
   RUNG wire#powerrail
      P_Contact(operand := "DISPARO_DIFERENCIAL_3Q3", bit := "MBIT_DISP_DIF_3Q3")
   END_RUNG wire#w1
   RUNG wire#powerrail
      P_Contact(operand := "DISPARO_DIFERENCIAL_4Q1_4Q2", bit := "MBIT_DISP_DIF_4Q1_4Q2")
   END_RUNG wire#w1
   RUNG wire#powerrail
      N_Contact(operand := "FALHA_24VDC", bit := "MBIT_FALHA_24VDC")
   END_RUNG wire#w1
   RUNG wire#powerrail
      P_Contact(operand := "FALHA_220VAC", bit := "MBIT_FALHA_220VAC")
   END_RUNG wire#w1
   RUNG wire#powerrail
      P_Contact(operand := "FALHA_24VAC", bit := "MBIT_FALHA_24VAC")
   END_RUNG wire#w1
   // the same network as SCL:
   #_w1 := "BS001A_DISPARO" AND NOT "MBIT_DISP_1";   // rising edge of "BS001A_DISPARO"
   "MBIT_DISP_1" := "BS001A_DISPARO";
   #_w2 := "BS001B_DISPARO" AND NOT "MBIT_DISP_2";   // rising edge of "BS001B_DISPARO"
   "MBIT_DISP_2" := "BS001B_DISPARO";
   #_w3 := "MX201_DISPARO" AND NOT "MBIT_DISP_3";   // rising edge of "MX201_DISPARO"
   "MBIT_DISP_3" := "MX201_DISPARO";
   #_w4 := "BH201_DISPARO" AND NOT "MBIT_DISP_4";   // rising edge of "BH201_DISPARO"
   "MBIT_DISP_4" := "BH201_DISPARO";
   #_w5 := "MX301_DISPARO" AND NOT "MBIT_DISP_5";   // rising edge of "MX301_DISPARO"
   "MBIT_DISP_5" := "MX301_DISPARO";
   #_w6 := "BM401_DISPARO" AND NOT "MBIT_DISP_6";   // rising edge of "BM401_DISPARO"
   "MBIT_DISP_6" := "BM401_DISPARO";
   #_w7 := "BS501_DISPARO" AND NOT "MBIT_DISP_7";   // rising edge of "BS501_DISPARO"
   "MBIT_DISP_7" := "BS501_DISPARO";
   #_w8 := "MX601_DISPARO" AND NOT "MBIT_DISP_8";   // rising edge of "MX601_DISPARO"
   "MBIT_DISP_8" := "MX601_DISPARO";
   #_w9 := "BD601_DISPARO" AND NOT "MBIT_DISP_9";   // rising edge of "BD601_DISPARO"
   "MBIT_DISP_9" := "BD601_DISPARO";
   #_w10 := "BD602_DISPARO" AND NOT "MBIT_DISP_10";   // rising edge of "BD602_DISPARO"
   "MBIT_DISP_10" := "BD602_DISPARO";
   #_w11 := "MX603_DISPARO" AND NOT "MBIT_DISP_11";   // rising edge of "MX603_DISPARO"
   "MBIT_DISP_11" := "MX603_DISPARO";
   #_w12 := "BD603_DISPARO" AND NOT "MBIT_DISP_12";   // rising edge of "BD603_DISPARO"
   "MBIT_DISP_12" := "BD603_DISPARO";
   #_w13 := "MX604_DISPARO" AND NOT "MBIT_DISP_13";   // rising edge of "MX604_DISPARO"
   "MBIT_DISP_13" := "MX604_DISPARO";
   #_w14 := "BD604_DISPARO" AND NOT "MBIT_DISP_14";   // rising edge of "BD604_DISPARO"
   "MBIT_DISP_14" := "BD604_DISPARO";
   #_w15 := "MX605_DISPARO" AND NOT "MBIT_DISP_15";   // rising edge of "MX605_DISPARO"
   "MBIT_DISP_15" := "MX605_DISPARO";
   #_w16 := "BD605_DISPARO" AND NOT "MBIT_DISP_16";   // rising edge of "BD605_DISPARO"
   "MBIT_DISP_16" := "BD605_DISPARO";
   #_w17 := "DISPARO_DIF_3Q1_32" AND NOT "MBIT_DISP_DIF_3Q1_32";   // rising edge of "DISPARO_DIF_3Q1_32"
   "MBIT_DISP_DIF_3Q1_32" := "DISPARO_DIF_3Q1_32";
   #_w18 := "DISPARO_DIFERENCIAL_3Q3" AND NOT "MBIT_DISP_DIF_3Q3";   // rising edge of "DISPARO_DIFERENCIAL_3Q3"
   "MBIT_DISP_DIF_3Q3" := "DISPARO_DIFERENCIAL_3Q3";
   #_w19 := "DISPARO_DIFERENCIAL_4Q1_4Q2" AND NOT "MBIT_DISP_DIF_4Q1_4Q2";   // rising edge of "DISPARO_DIFERENCIAL_4Q1_4Q2"
   "MBIT_DISP_DIF_4Q1_4Q2" := "DISPARO_DIFERENCIAL_4Q1_4Q2";
   #_w20 := NOT "FALHA_24VDC" AND "MBIT_FALHA_24VDC";   // falling edge of "FALHA_24VDC"
   "MBIT_FALHA_24VDC" := "FALHA_24VDC";
   #_w21 := "FALHA_220VAC" AND NOT "MBIT_FALHA_220VAC";   // rising edge of "FALHA_220VAC"
   "MBIT_FALHA_220VAC" := "FALHA_220VAC";
   #_w22 := "FALHA_24VAC" AND NOT "MBIT_FALHA_24VAC";   // rising edge of "FALHA_24VAC"
   "MBIT_FALHA_24VAC" := "FALHA_24VAC";
   "Alarmes".ALARME_DISPARO := #_w1 OR #_w2 OR #_w3 OR #_w4 OR #_w5 OR #_w6 OR #_w7 OR #_w8 OR #_w9 OR #_w10 OR #_w11 OR #_w12 OR #_w13 OR #_w14 OR #_w15 OR #_w16 OR #_w17 OR #_w18 OR #_w19 OR #_w20 OR #_w21 OR #_w22;
END_REGION
END_FUNCTION

FUNCTION "Alarmes_Disparos_2" : Void
{ S7_Optimized_Access := 'TRUE' }
VERSION : 0.1

BEGIN
	"Alarmes".ALARMES_1.%X3 := "BS001A_DISPARO";
	"Alarmes".ALARMES_1.%X4 := "BS001B_DISPARO";
	"Alarmes".ALARMES_1.%X5 := "MX201_DISPARO";
	"Alarmes".ALARMES_1.%X6 := "BH201_DISPARO";
	"Alarmes".ALARMES_1.%X7 := "MX301_DISPARO";
	"Alarmes".ALARMES_1.%X8 := "BM401_DISPARO";
	"Alarmes".ALARMES_1.%X9 := "BS501_DISPARO";
	"Alarmes".ALARMES_1.%X10 := "MX601_DISPARO";
	"Alarmes".ALARMES_1.%X11 := "BD601_DISPARO";
	"Alarmes".ALARMES_1.%X12 := "BD602_DISPARO";
	"Alarmes".ALARMES_1.%X13 := "MX603_DISPARO";
	"Alarmes".ALARMES_1.%X14 := "BD603_DISPARO";
	"Alarmes".ALARMES_1.%X15 := "MX604_DISPARO";
	"Alarmes".ALARMES_2.%X0 := "BD604_DISPARO";
	"Alarmes".ALARMES_2.%X1 := "MX605_DISPARO";
	"Alarmes".ALARMES_2.%X2 := "BD605_DISPARO";
	"Alarmes".ALARMES_2.%X3 := "DISPARO_DIF_3Q1_32";
	"Alarmes".ALARMES_2.%X4 := "DISPARO_DIFERENCIAL_3Q3";
	"Alarmes".ALARMES_2.%X5 := "DISPARO_DIFERENCIAL_4Q1_4Q2";
	"Alarmes".ALARMES_2.%X6 := NOT "FALHA_24VDC";
	"Alarmes".ALARMES_2.%X7 := "FALHA_220VAC";
	"Alarmes".ALARMES_2.%X8 := "FALHA_24VAC";
	
	
	
	
	
	
	
	
	
	
	
	
	
	
	
END_FUNCTION

FUNCTION "Alarme_XV102" : Void   // FC24, LAD
{ S7_Optimized_Access := 'TRUE' }
VERSION : 0.1
// stored: AutoNumber true, IsIECCheckEnabled false, SetENOAutomatically false, UDAEnableTagReadback false
BEGIN

REGION Network 1: XV102 a abrir
